# B&R Automation Studio project PT_KB_V01
Automation Studio 4.12.3.127 SP

## Configuration C50_Terminal

CPU 4PPC50.101E-13A, AutomationRuntime B4.93, Build 4.1.2, Vc V4.73.3

### Hardware
```
4PPC50_101E_13A : 4PPC50.101E-13A v1.2.2.0
  Connector IF2:
    ActivateDevice = 1
    Mode = Manual
    InternetAddress = 10.0.0.205
    SubnetMask = 255.255.254.0
  Connector IF3:
    AssignedOperatingSystem = ARemb
  Connector IF4:
    AssignedOperatingSystem = GPOS
  ConfigurationID = PT_KB_V01_C50_Terminal
  TimerDeviceType = SWIOTIMER
  Cyclic1Duration = 10000
  Cyclic1Tolerance = 10000
  Cyclic2Duration = 20000
  Cyclic2Tolerance = 20000
  Cyclic3Duration = 50000
  Cyclic3Tolerance = 50000
  Cyclic4Duration = 100000
  Cyclic4Tolerance = 100000
  Cyclic5Duration = 200000
  Cyclic5Tolerance = 200000
  Cyclic6Duration = 500000
  Cyclic6Tolerance = 500000
  Cyclic7Duration = 1000000
  Cyclic7Tolerance = 1000000
  Cyclic8Duration = 10000
  Cyclic8Tolerance = 30000000
  FileDevice1
  FileDeviceName1 = USER
  FileDevicePath1 = USER_PATH
  LXTMode = Manual
  LXTInternetAddress = 10.0.0.205
  LXTSubnetmask = 255.255.254.0
  LXTActivateDns = 0
  LXTVisuMode = VNC
  LXTVisuURL = 10.0.0.204:5900
  LXTPasswordVNC = 
  LXTUpdateTrigger = 0
```

## Configuration Config1

CPU 4PPC50.101E-13A, AutomationRuntime B4.93, Build 4.1.2, Vc V4.73.3

### Task classes (Cpu.sw)
```
Cyclic#1 (cycle 10000 us, tolerance 10000 us):
  IO <- IO.prg
Cyclic#4 (cycle 100000 us, tolerance 100000 us):
  PID_Pu_01 <- PID_Pu_01.prg
  Rad_PG_KB <- Rad_PG_KB.prg
  PG_Intf <- PG_Intf.prg
  HMI_Svc <- HMI_Svc.prg
  ProcUnit <- ProcessUnit.ProcUnit.prg
  DeviceCtrl <- DeviceCtrl.prg
Cyclic#5 (cycle 200000 us, tolerance 200000 us):
  BRB2_com <- IMA_comm_PG_BRB2.BRB2_com.prg
DataObjects: BRB2 <- IMA_comm_PG_BRB2.BRB2.dob
VcDataObjects: Visu1 <- Visu1.dob
Binaries: vcmgr, arialbd, udbdef, vcpdsw, vcalarm, vcshared, vcgclass, Visu101, vctcal, vccshape, vcnet, TCData, vcpdvnc, vcctext, FWRules, vcdsint, vcfile, Visu102, vcrt, vcbclass, vcpfgen, vcfntttf, vcdsloc, vccovl, Visu103, arial, vccnum, vccstr, vccbtn, ashwd, ashwac, User, sysconf, asfw, arconfig, iomap, Role
Libraries: standard, MTBasics, brsystem, sys_lib, MTTypes, runtime, MTFilter, FileIO, AsArLog, AsArProf, AsMem, DataObj, astime, BR_Lib, VFD_Lib, vcresman, asieccon, AsIMA, inaclnt
```

### Hardware
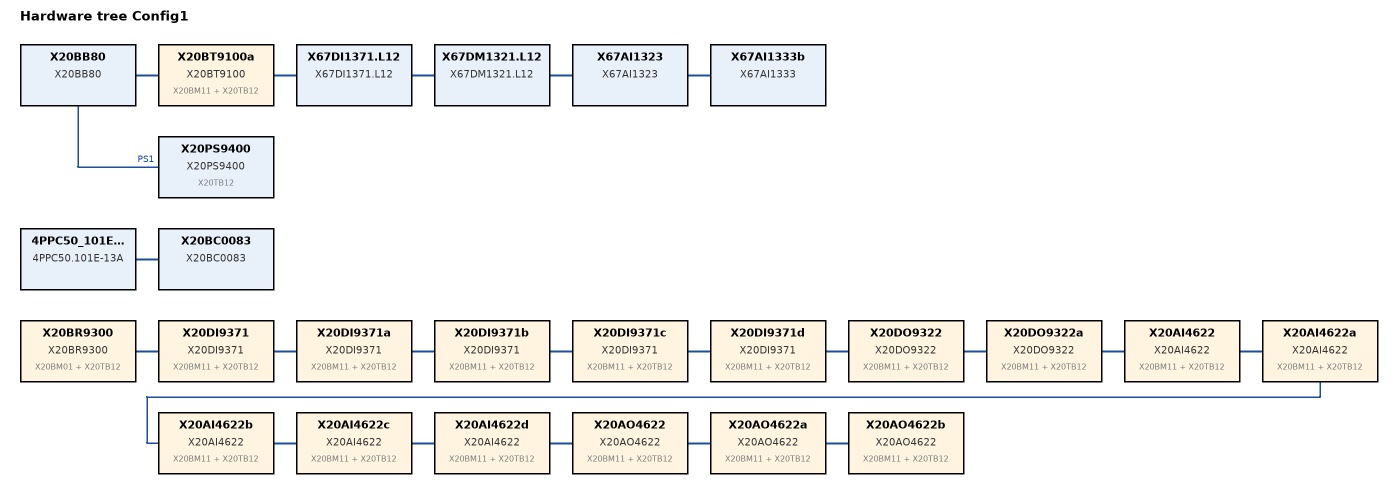
```
4PPC50_101E_13A : 4PPC50.101E-13A v1.2.2.0
  Connector IF2:
    ActivateDevice = 1
    Mode = Manual
    InternetAddress = 10.0.0.204
    SubnetMask = 255.255.254.0
  Connector IF3:
    AssignedOperatingSystem = ARemb
  Connector IF4:
    AssignedOperatingSystem = GPOS
  ConfigurationID = PT_KB_V01_Config1
  RemanentGlobalPvSize = 5000
  VolatileGlobalPvSize = 655350
  RebootReset = 1
  TimerDeviceType = SWIOTIMER
  Cyclic1Duration = 10000
  Cyclic1Tolerance = 10000
  Cyclic2Duration = 20000
  Cyclic2Tolerance = 20000
  Cyclic3Duration = 50000
  Cyclic3Tolerance = 50000
  Cyclic4Duration = 100000
  Cyclic4Tolerance = 100000
  Cyclic5Duration = 200000
  Cyclic5Tolerance = 200000
  Cyclic6Duration = 500000
  Cyclic6Tolerance = 500000
  Cyclic7Duration = 1000000
  Cyclic7Tolerance = 1000000
  Cyclic8Duration = 10000
  Cyclic8Tolerance = 30000000
  FileDevice1
  FileDeviceName1 = USER
  FileDevicePath1 = USER_PATH
  VncVcObjectName = Visu1
  VncMaxConnections = 5
  LXTMode = Manual
  LXTInternetAddress = 10.0.0.205
  LXTSubnetmask = 255.255.254.0
  LXTActivateBuzzer = 1
  LXTVisuMode = VNC
  LXTVisuURL = 10.0.0.204:5900
  LXTPasswordVNC = 
  LXTLocalScaling = 1
  LXTUpdateTrigger = 0
X20AI4622 : X20AI4622 v1.5.0.0  [SS1 -> X20TB12h.SS; SL -> X20BM11g.SL1]
  ChannelType01 = 4 to 20mA
  ChannelType02 = 4 to 20mA
  ChannelType03 = 4 to 20mA
  ChannelType04 = 4 to 20mA
X20AI4622a : X20AI4622 v1.5.0.0  [SS1 -> X20TB12i.SS; SL -> X20BM11h.SL1]
  ChannelType01 = 4 to 20mA
  ChannelType02 = 4 to 20mA
  ChannelType03 = 4 to 20mA
  ChannelType04 = 4 to 20mA
X20AI4622b : X20AI4622 v1.5.0.0  [SS1 -> X20TB12j.SS; SL -> X20BM11i.SL1]
  ChannelType01 = 4 to 20mA
  ChannelType02 = 4 to 20mA
  ChannelType03 = 4 to 20mA
  ChannelType04 = 4 to 20mA
X20AI4622c : X20AI4622 v1.5.0.0  [SS1 -> X20TB12k.SS; SL -> X20BM11j.SL1]
  ChannelType01 = 4 to 20mA
  ChannelType02 = 4 to 20mA
  ChannelType03 = 4 to 20mA
  ChannelType04 = 4 to 20mA
X20AI4622d : X20AI4622 v1.5.0.0  [SS1 -> X20TB12l.SS; SL -> X20BM11k.SL1]
  ChannelType01 = 4 to 20mA
  ChannelType02 = 4 to 20mA
  ChannelType03 = 4 to 20mA
  ChannelType04 = 4 to 20mA
X20AO4622 : X20AO4622 v1.4.1.0  [SS1 -> X20TB12m.SS; SL -> X20BM11l.SL1]
  ChannelType01 = 4 to 20mA
  ChannelType02 = 4 to 20mA
  ChannelType03 = 4 to 20mA
  ChannelType04 = 4 to 20mA
X20AO4622a : X20AO4622 v1.4.1.0  [SS1 -> X20TB12n.SS; SL -> X20BM11m.SL1]
  ChannelType01 = 4 to 20mA
  ChannelType02 = 4 to 20mA
  ChannelType03 = 4 to 20mA
  ChannelType04 = 4 to 20mA
X20AO4622b : X20AO4622 v1.4.1.0  [SS1 -> X20TB12o.SS; SL -> X20BM11n.SL1]
  ChannelType01 = 4 to 20mA
  ChannelType02 = 4 to 20mA
  ChannelType03 = 4 to 20mA
  ChannelType04 = 4 to 20mA
X20BB80 : X20BB80 v1.1.0.0
X20BC0083 : X20BC0083 v2.14.0.0  [PLK1 -> 4PPC50_101E_13A.IF1 (NodeNumber=16) [Cable Type=PowerlinkCable, Length=10, Version=1.0.0.3]; SL -> X20BB80.SL1]
  Supervision = off
X20BM01 : X20BM01 v2.2.0.0
X20BM11 : X20BM11 v1.1.0.0  [X2X1 -> X20BM01.X2X2]
X20BM11a : X20BM11 v1.1.0.0  [X2X1 -> X20BM11.X2X2]
X20BM11b : X20BM11 v1.1.0.0  [X2X1 -> X20BM11a.X2X2]
X20BM11c : X20BM11 v1.1.0.0  [X2X1 -> X20BM11b.X2X2]
X20BM11d : X20BM11 v1.1.0.0  [X2X1 -> X20BM11c.X2X2]
X20BM11e : X20BM11 v1.1.0.0  [X2X1 -> X20BM11d.X2X2]
X20BM11f : X20BM11 v1.1.0.0  [X2X1 -> X20BM11e.X2X2]
X20BM11g : X20BM11 v1.1.0.0  [X2X1 -> X20BM11f.X2X2]
X20BM11h : X20BM11 v1.1.0.0  [X2X1 -> X20BM11g.X2X2]
X20BM11i : X20BM11 v1.1.0.0  [X2X1 -> X20BM11h.X2X2]
X20BM11j : X20BM11 v1.1.0.0  [X2X1 -> X20BM11i.X2X2]
X20BM11k : X20BM11 v1.1.0.0  [X2X1 -> X20BM11j.X2X2]
X20BM11l : X20BM11 v1.1.0.0  [X2X1 -> X20BM11k.X2X2]
X20BM11m : X20BM11 v1.1.0.0  [X2X1 -> X20BM11l.X2X2]
X20BM11n : X20BM11 v1.1.0.0  [X2X1 -> X20BM11m.X2X2]
X20BM11p : X20BM11 v1.1.0.0  [X2X1 -> X20BB80.IF1]
X20BR9300 : X20BR9300 v1.3.0.0  [SS1 -> X20TB12.SS; SL -> X20BM01.SL1; X2X1 -> 4PPC50_101E_13A.IF5 [Cable Type=X2XCable, Length=10, Version=1.0.0.3]]
X20BT9100a : X20BT9100 v1.3.0.0  [SS1 -> X20TB12q.SS; SL -> X20BM11p.SL1]
X20DI9371 : X20DI9371 v1.6.0.0  [SS1 -> X20TB12a.SS; SL -> X20BM11.SL1]
X20DI9371a : X20DI9371 v1.6.0.0  [SS1 -> X20TB12b.SS; SL -> X20BM11a.SL1]
X20DI9371b : X20DI9371 v1.6.0.0  [SS1 -> X20TB12c.SS; SL -> X20BM11b.SL1]
X20DI9371c : X20DI9371 v1.6.0.0  [SS1 -> X20TB12d.SS; SL -> X20BM11c.SL1]
X20DI9371d : X20DI9371 v1.6.0.0  [SS1 -> X20TB12e.SS; SL -> X20BM11d.SL1]
X20DO9322 : X20DO9322 v1.6.0.0  [SS1 -> X20TB12f.SS; SL -> X20BM11e.SL1]
X20DO9322a : X20DO9322 v1.6.0.0  [SS1 -> X20TB12g.SS; SL -> X20BM11f.SL1]
X20PS9400 : X20PS9400 v1.8.0.0  [SS1 -> X20TB12r.SS; PS -> X20BB80.PS1]
X20TB12 : X20TB12 v1.0.0.0
X20TB12a : X20TB12 v1.0.0.0
X20TB12b : X20TB12 v1.0.0.0
X20TB12c : X20TB12 v1.0.0.0
X20TB12d : X20TB12 v1.0.0.0
X20TB12e : X20TB12 v1.0.0.0
X20TB12f : X20TB12 v1.0.0.0
X20TB12g : X20TB12 v1.0.0.0
X20TB12h : X20TB12 v1.0.0.0
X20TB12i : X20TB12 v1.0.0.0
X20TB12j : X20TB12 v1.0.0.0
X20TB12k : X20TB12 v1.0.0.0
X20TB12l : X20TB12 v1.0.0.0
X20TB12m : X20TB12 v1.0.0.0
X20TB12n : X20TB12 v1.0.0.0
X20TB12o : X20TB12 v1.0.0.0
X20TB12q : X20TB12 v1.0.0.0
X20TB12r : X20TB12 v1.0.0.0
X67AI1323 : X67AI1323 v1.1.0.0  [X2X1 -> X67DM1321.L12.X2X2 [Cable Type=X2XCable, Length=10, Version=1.0.0.3]]
  Supervision = off
  InputFilter = level 128
  EnhChannelConfig = on
  ChannelType01 = 4to20mA
  ChannelType02 = 4to20mA
  ChannelType03 = 4to20mA
  ChannelType04 = 4to20mA
X67AI1333b : X67AI1333 v1.1.0.0  [X2X1 -> X67AI1323.X2X2 [Cable Type=X2XCable, Length=10, Version=1.0.0.3]]
  Supervision = off
  InputFilter = level 128
  ChannelType01 = 4to20mA
  ChannelType02 = 4to20mA
  ChannelType03 = 4to20mA
  ChannelType04 = 4to20mA
X67DI1371.L12 : X67DI1371.L12 v1.1.0.0  [X2X1 -> X20BT9100a.X2X1 [Cable Type=X2XCable, Length=10, Version=1.0.0.3]]
  Supervision = off
X67DM1321.L12 : X67DM1321.L12 v1.3.0.0  [X2X1 -> X67DI1371.L12.X2X2 [Cable Type=X2XCable, Length=10, Version=1.0.0.3]]
  Supervision = off
```

### IoMap.iom - 4PPC50_101E_13A/IoMap.iom
```iecst
VAR_CONFIG
	Cyclic#1.PG.Sens.Pt._1.AI_Input.RawValue AT %IW."X20AI4622".AnalogInput01; (* PT01 - pritisak termalne vode na ulazu podstanice [bar]. *)
	Cyclic#1.PG.Sens.Pt._2.AI_Input.RawValue AT %IW."X20AI4622".AnalogInput02; (* PT02 - pritisak posle streinera grubih filtera [bar]. *)
	Cyclic#1.PG.Sens.Pt._3.AI_Input.RawValue AT %IW."X20AI4622".AnalogInput03; (* PT03 - pritisak posle velikog razmenjivaca [bar]. *)
	Cyclic#1.PG.Sens.Pt._4.AI_Input.RawValue AT %IW."X20AI4622".AnalogInput04; (* PT04 - pritisak na ulazu u prihvatni tank [bar]. *)
	Cyclic#1.PG.Sens.Pt._5.AI_Input.RawValue AT %IW."X20AI4622a".AnalogInput01; (* PT05 - pritisak na potisu transportnih pumpi [bar]. *)
	Cyclic#1.PG.Sens.Pt._NS1.AI_Input.RawValue AT %IW."X20AI4622a".AnalogInput02; (* PTNS01 - pritisak na dnu prihvatnog tanka [bar]. *)
	Cyclic#1.PG.Sens.Pt._NS2.AI_Input.RawValue AT %IW."X20AI4622a".AnalogInput03; (* PTNS02 - pritisak na vrhu prihvatnog tanka [bar]. *)
	Cyclic#1.PG.Sens.Pt._0_0.AI_Input.RawValue AT %IW."X20AI4622a".AnalogInput04; (* Pritisak komprimovanog vazduha [bar]. *)
	Cyclic#1.PG.Sens.Tt._7.AI_Input.RawValue AT %IW."X20AI4622b".AnalogInput01;
	Cyclic#1.PG.Sens.Tt._2.AI_Input.RawValue AT %IW."X20AI4622b".AnalogInput02; (* TT_PG_02 - ulaz u prihvatni tank. *)
	Cyclic#1.PG.Sens.Tt._3.AI_Input.RawValue AT %IW."X20AI4622b".AnalogInput03; (* TT_PG_03 - temperatura u prihvatnom tanku. *)
	Cyclic#1.PG.Act.PV._5.PV_Input.AI_Raw AT %IW."X20AI4622b".AnalogInput04; (* PG_PV05 - analogna povratna pozicija ventila. *)
	Cyclic#1.PG.Sens.MP._1.AI_Input.RawValue AT %IW."X20AI4622c".AnalogInput01; (* MP01 - protok potisa ka potrosacima [l/s]. *)
	Cyclic#1.PG.Sens.Pt._6.AI_Input.RawValue AT %IW."X20AI4622c".AnalogInput02; (* PT06 - dodatni transmiter pritiska [bar]. *)
	Cyclic#1.PG.Act.PV._1.PV_Input.AI_Raw AT %IW."X20AI4622d".AnalogInput01; (* PG_PV01 - analogna povratna pozicija ulaznog ventila tanka. *)
	Cyclic#1.PG.Act.PV._2.PV_Input.AI_Raw AT %IW."X20AI4622d".AnalogInput02; (* PG_PV02 - analogna povratna pozicija ulaznog ventila tanka. *)
	Cyclic#1.PG.Act.PV._3.PV_Input.AI_Raw AT %IW."X20AI4622d".AnalogInput03; (* PV03 - analogna povratna pozicija odzracnog ventila ulaza podstanice. *)
	Cyclic#1.PG.Act.PV._4.PV_Input.AI_Raw AT %IW."X20AI4622d".AnalogInput04; (* PV04 - analogna povratna pozicija odzracnog ventila ulaza tanka. *)
	Cyclic#1.PG.Act.Pu._1.mapping.DIO.w_freq AT %QW."X20AO4622".AnalogOutput01; (* PG_Pu01 - frekventni zahtev VFD-a [procenat opsega]. *)
	Cyclic#1.PG.Act.Pu._2.mapping.DIO.w_freq AT %QW."X20AO4622".AnalogOutput02; (* PG_Pu02 - frekventni zahtev VFD-a [procenat opsega]. *)
	Cyclic#1.PG.Act.PV._1.PV_Output.AO_Raw AT %QW."X20AO4622a".AnalogOutput01; (* PG_PV01 - analogna komanda polozaja ulaznog ventila tanka. *)
	Cyclic#1.PG.Act.PV._2.PV_Output.AO_Raw AT %QW."X20AO4622a".AnalogOutput02; (* PG_PV02 - analogna komanda polozaja ulaznog ventila tanka. *)
	Cyclic#1.PG.Act.PV._3.PV_Output.AO_Raw AT %QW."X20AO4622a".AnalogOutput03; (* PV03 - analogna komanda polozaja odzracnog ventila ulaza podstanice. *)
	Cyclic#1.PG.Act.PV._4.PV_Output.AO_Raw AT %QW."X20AO4622a".AnalogOutput04; (* PV04 - analogna komanda polozaja odzracnog ventila ulaza tanka. *)
	Cyclic#1.PG.Act.PV._5.PV_Output.AO_Raw AT %QW."X20AO4622b".AnalogOutput01; (* PG_PV05 - analogna komanda polozaja ventila drenaze/preispiranja. *)
	Cyclic#1.PG.Act.Pu._1.mapping.DIO.r_error AT %IX."X20DI9371".DigitalInput01; (* PG_Pu01 - fault ulaz frekventnog regulatora. *)
	Cyclic#1.PG.Act.Pu._2.mapping.DIO.r_error AT %IX."X20DI9371".DigitalInput02; (* PG_Pu02 - fault ulaz frekventnog regulatora. *)
	Cyclic#1.PG.Act.AV._1.V_Input.CloseFb AT %IX."X20DI9371".DigitalInput03; (* PG_V01 - potvrdjen zatvoren polozaj IEBKB1 dovoda. *)
	Cyclic#1.PG.Act.AV._1.V_Input.OpenFb AT %IX."X20DI9371".DigitalInput04; (* PG_V01 - potvrdjen otvoren polozaj IEBKB1 dovoda. *)
	Cyclic#1.PG.Act.AV._2.V_Input.CloseFb AT %IX."X20DI9371".DigitalInput05; (* PG_V02 - potvrdjen zatvoren polozaj BRB2 dovoda. *)
	Cyclic#1.PG.Act.AV._2.V_Input.OpenFb AT %IX."X20DI9371".DigitalInput06; (* PG_V02 - potvrdjen otvoren polozaj BRB2 dovoda. *)
	Cyclic#1.PG.Act.RV._25.HV_Input.CloseFb AT %IX."X20DI9371b".DigitalInput05; (* PG_RV25 - rucni gasni bypass iz tanka, zatvoren. *)
	Cyclic#1.PG.Act.RV._25.HV_Input.OpenFb AT %IX."X20DI9371b".DigitalInput06; (* PG_RV25 - rucni gasni bypass iz tanka, otvoren. *)
	Cyclic#1.PG.Act.RV._26.HV_Input.CloseFb AT %IX."X20DI9371b".DigitalInput07; (* PG_RV26 - rucni ulazni ventil vakuum pumpe, zatvoren. *)
	Cyclic#1.PG.Act.RV._26.HV_Input.OpenFb AT %IX."X20DI9371b".DigitalInput08; (* PG_RV26 - rucni ulazni ventil vakuum pumpe, otvoren. *)
	Cyclic#1.PG.Act.RV._27.HV_Input.CloseFb AT %IX."X20DI9371b".DigitalInput09; (* PG_RV27 - rucni izlazni ventil vakuum pumpe, zatvoren. *)
	Cyclic#1.PG.Act.RV._27.HV_Input.OpenFb AT %IX."X20DI9371b".DigitalInput10; (* PG_RV27 - rucni izlazni ventil vakuum pumpe, otvoren. *)
	Cyclic#1.PG.Sens.LS._1.DI_Input.SensorIn AT %IX."X20DI9371c".DigitalInput01; (* LS01 - nizak nivo prihvatnog tanka. *)
	Cyclic#1.PG.Sens.LS._2.DI_Input.SensorIn AT %IX."X20DI9371c".DigitalInput02; (* LS02 - donji nivo odzracnog cilindra na ulazu podstanice. *)
	Cyclic#1.PG.Sens.LS._3.DI_Input.SensorIn AT %IX."X20DI9371c".DigitalInput03; (* LS03 - gornji nivo odzracnog cilindra na ulazu podstanice. *)
	Cyclic#1.PG.Sens.LS._4.DI_Input.SensorIn AT %IX."X20DI9371c".DigitalInput04; (* LS04 - donji nivo odzracnog cilindra na ulazu tanka. *)
	Cyclic#1.PG.Sens.LS._5.DI_Input.SensorIn AT %IX."X20DI9371c".DigitalInput05; (* LS05 - gornji nivo odzracnog cilindra na ulazu tanka. *)
	Cyclic#1.PG.Sens.MP._1.AI_Input.TransmitterStatus AT %IX."X20DI9371c".DigitalInput06; (* MP01 - status meraca protoka potisa ka potrosacima. *)
	Cyclic#1.PG.Act.AV._1.V_Input.LampOpen AT %IX."X20DI9371c".DigitalInput07; (* PG_V01 - signal pogona dostigao otvoren kraj. *)
	Cyclic#1.PG.Act.AV._1.V_Input.LampClose AT %IX."X20DI9371c".DigitalInput08; (* PG_V01 - signal pogona dostigao zatvoren kraj. *)
	Cyclic#1.PG.Act.AV._2.V_Input.LampOpen AT %IX."X20DI9371c".DigitalInput09; (* PG_V02 - signal pogona dostigao otvoren kraj. *)
	Cyclic#1.PG.Act.AV._2.V_Input.LampClose AT %IX."X20DI9371c".DigitalInput10; (* PG_V02 - signal pogona dostigao zatvoren kraj. *)
	Cyclic#1.PG.Act.AV._1.V_Input.OverTorque AT %IX."X20DI9371c".DigitalInput11; (* PG_V01 - zastita pogona od prevelikog momenta. *)
	Cyclic#1.PG.Act.Pu._1.mapping.DIO.w_run_fwd AT %QX."X20DO9322".DigitalOutput01; (* PG_Pu01 - komanda rad napred. *)
	Cyclic#1.PG.Act.Pu._1.mapping.DIO.w_reset AT %QX."X20DO9322".DigitalOutput02; (* PG_Pu01 - komanda reset greske pogona. *)
	Cyclic#1.PG.Act.Pu._2.mapping.DIO.w_run_fwd AT %QX."X20DO9322".DigitalOutput03; (* PG_Pu02 - komanda rad napred. *)
	Cyclic#1.PG.Act.Pu._2.mapping.DIO.w_reset AT %QX."X20DO9322".DigitalOutput04; (* PG_Pu02 - komanda reset greske pogona. *)
	Cyclic#1.PG.Act.AV._1.V_Output.CmdOpen AT %QX."X20DO9322".DigitalOutput05; (* PG_V01 - komanda otvaranja bistabilnog IEBKB1 dovoda. *)
	Cyclic#1.PG.Act.AV._1.V_Output.CmdClose AT %QX."X20DO9322".DigitalOutput06; (* PG_V01 - komanda zatvaranja bistabilnog IEBKB1 dovoda. *)
	Cyclic#1.PG.Act.AV._2.V_Output.CmdOpen AT %QX."X20DO9322".DigitalOutput07; (* PG_V02 - komanda otvaranja bistabilnog BRB2 dovoda. *)
	Cyclic#1.PG.Act.AV._2.V_Output.CmdClose AT %QX."X20DO9322".DigitalOutput08; (* PG_V02 - komanda zatvaranja bistabilnog BRB2 dovoda. *)
	Cyclic#1.PG.Act.AV._3.V_Output.Cmd AT %QX."X20DO9322".DigitalOutput09; (* PG_V03 - komanda otvaranja pneumatskog ventila izlaza PG_Pu01. *)
	Cyclic#1.PG.Act.AV._4.V_Output.Cmd AT %QX."X20DO9322".DigitalOutput10; (* PG_V04 - komanda otvaranja pneumatskog ventila izlaza PG_Pu02. *)
	Cyclic#1.PG.Act.AV._5.V_Output.Cmd AT %QX."X20DO9322".DigitalOutput11; (* PG_V05 - komanda otvaranja pneumatskog bypass ventila. *)
	Cyclic#1.PG.Act.AV._6.V_Output.Cmd AT %QX."X20DO9322".DigitalOutput12; (* PG_V06 - komanda otvaranja pneumatske grane PG_PV01. *)
	Cyclic#1.PG.Act.AV._7.V_Output.Cmd AT %QX."X20DO9322a".DigitalOutput01; (* PG_V07 - komanda otvaranja pneumatske grane PG_PV02. *)
	Cyclic#1.PG.Sens.Tt._5.AI_Input.RawValue AT %IW."X67AI1323".AnalogInput01;
	Cyclic#1.PG.Sens.Tt._6.AI_Input.RawValue AT %IW."X67AI1323".AnalogInput02;
	Cyclic#1.PG.Sens.Tt._10.AI_Input.RawValue AT %IW."X67AI1323".AnalogInput03;
	Cyclic#1.PG.Sens.Tt._11.AI_Input.RawValue AT %IW."X67AI1323".AnalogInput04;
	Cyclic#1.PG.Sens.Tt._1.AI_Input.RawValue AT %IW."X67AI1333b".AnalogInput01;
	Cyclic#1.PG.Sens.Tt._4.AI_Input.RawValue AT %IW."X67AI1333b".AnalogInput02;
	Cyclic#1.PG.Sens.Tt._9.AI_Input.RawValue AT %IW."X67AI1333b".AnalogInput03;
	Cyclic#1.PG.Sens.Tt._8.AI_Input.RawValue AT %IW."X67AI1333b".AnalogInput04;
	Cyclic#1.PG.Act.AV._3.V_Input.CloseFb AT %IX."X67DI1371.L12".DigitalInput01;
	Cyclic#1.PG.Act.AV._3.V_Input.OpenFb AT %IX."X67DI1371.L12".DigitalInput02;
	Cyclic#1.PG.Act.AV._4.V_Input.CloseFb AT %IX."X67DI1371.L12".DigitalInput03;
	Cyclic#1.PG.Act.AV._4.V_Input.OpenFb AT %IX."X67DI1371.L12".DigitalInput04;
	Cyclic#1.PG.Act.RV._22.HV_Input.CloseFb AT %IX."X67DI1371.L12".DigitalInput05;
	Cyclic#1.PG.Act.RV._22.HV_Input.OpenFb AT %IX."X67DI1371.L12".DigitalInput06;
	Cyclic#1.PG.Act.RV._23.HV_Input.CloseFb AT %IX."X67DI1371.L12".DigitalInput07;
	Cyclic#1.PG.Act.RV._23.HV_Input.OpenFb AT %IX."X67DI1371.L12".DigitalInput08;
	Cyclic#1.PG.Act.RV._24.HV_Input.CloseFb AT %IX."X67DI1371.L12".DigitalInput09;
	Cyclic#1.PG.Act.RV._24.HV_Input.OpenFb AT %IX."X67DI1371.L12".DigitalInput10;
	Cyclic#1.PG.Act.AV._5.V_Input.CloseFb AT %IX."X67DM1321.L12".DigitalInput01;
	Cyclic#1.PG.Act.AV._5.V_Input.OpenFb AT %IX."X67DM1321.L12".DigitalInput02;
	Cyclic#1.PG.Act.AV._6.V_Input.CloseFb AT %IX."X67DM1321.L12".DigitalInput03;
	Cyclic#1.PG.Act.AV._6.V_Input.OpenFb AT %IX."X67DM1321.L12".DigitalInput04;
	Cyclic#1.PG.Act.AV._7.V_Input.CloseFb AT %IX."X67DM1321.L12".DigitalInput05;
	Cyclic#1.PG.Act.AV._7.V_Input.OpenFb AT %IX."X67DM1321.L12".DigitalInput06;
	Cyclic#1.PG.Act.RV._19.HV_Input.CloseFb AT %IX."X67DM1321.L12".DigitalInput07;
	Cyclic#1.PG.Act.RV._19.HV_Input.OpenFb AT %IX."X67DM1321.L12".DigitalInput08;
	Cyclic#1.PG.Act.RV._21.HV_Input.CloseFb AT %IX."X67DM1321.L12".DigitalInput09;
	Cyclic#1.PG.Act.RV._21.HV_Input.OpenFb AT %IX."X67DM1321.L12".DigitalInput10;
	Cyclic#1.PG.Sens.OWF._1.DI_Input.SensorIn AT %IX."X67DM1321.L12".DigitalInput11;
	Cyclic#1.PG.Sens.OWF._2.DI_Input.SensorIn AT %IX."X67DM1321.L12".DigitalInput12;
END_VAR
```

## Configuration Config2

CPU X20CP1382, AutomationRuntime I4.83, Build 4.1.2, Vc V4.73.0

### Task classes (Cpu.sw)
```
Cyclic#1:
  IO <- Project.IO.prg
Cyclic#4:
  Rad_PG_KB <- Project.Rad_PG_KB.prg
  PID_Pu_PT <- Project.PID_Pu_PT.prg
  PG_Intf <- Project.PG_Intf.prg
  HMI_Svc <- Project.HMI_Svc.prg
  ProcUnit <- ProcessUnit.ProcUnit.prg
  DeviceCtrl <- Project.DeviceCtrl.prg
  Cfg2ATV <- CAN.prg
Cyclic#5:
  BRB2_com <- IMA_comm_PG_BRB2.BRB2_com.prg
DataObjects: BRB2 <- IMA_comm_PG_BRB2.BRB2.dob
VcDataObjects: PG1_1 <- Project.PG1_1.dob
Binaries: vcmgr, arialbd, udbdef, vcpdsw, vcalarm, vcshared, vcgclass, Visu101, vctcal, vccshape, vcnet, TCData, vcpdvnc, vcctext, FWRules, vcdsint, vcfile, Visu102, vcrt, vcbclass, vcfntttf, vcdsloc, vccovl, Visu103, arial, vccnum, vccstr, vccbtn, vcpkat, vccdt, vccline, vcctrend, vccbar, vcpfx20, ashwd, ashwac, User, sysconf, asfw, arconfig, iomap, Role, vcpfgen
Libraries: standard, MTBasics, brsystem, sys_lib, MTTypes, runtime, MTFilter, FileIO, AsArLog, AsArProf, AsMem, DataObj, astime, BR_Lib, VFD_Lib, NashCan1, AsIMA, inaclnt, vcresman, asieccon, ashw
```

### Hardware
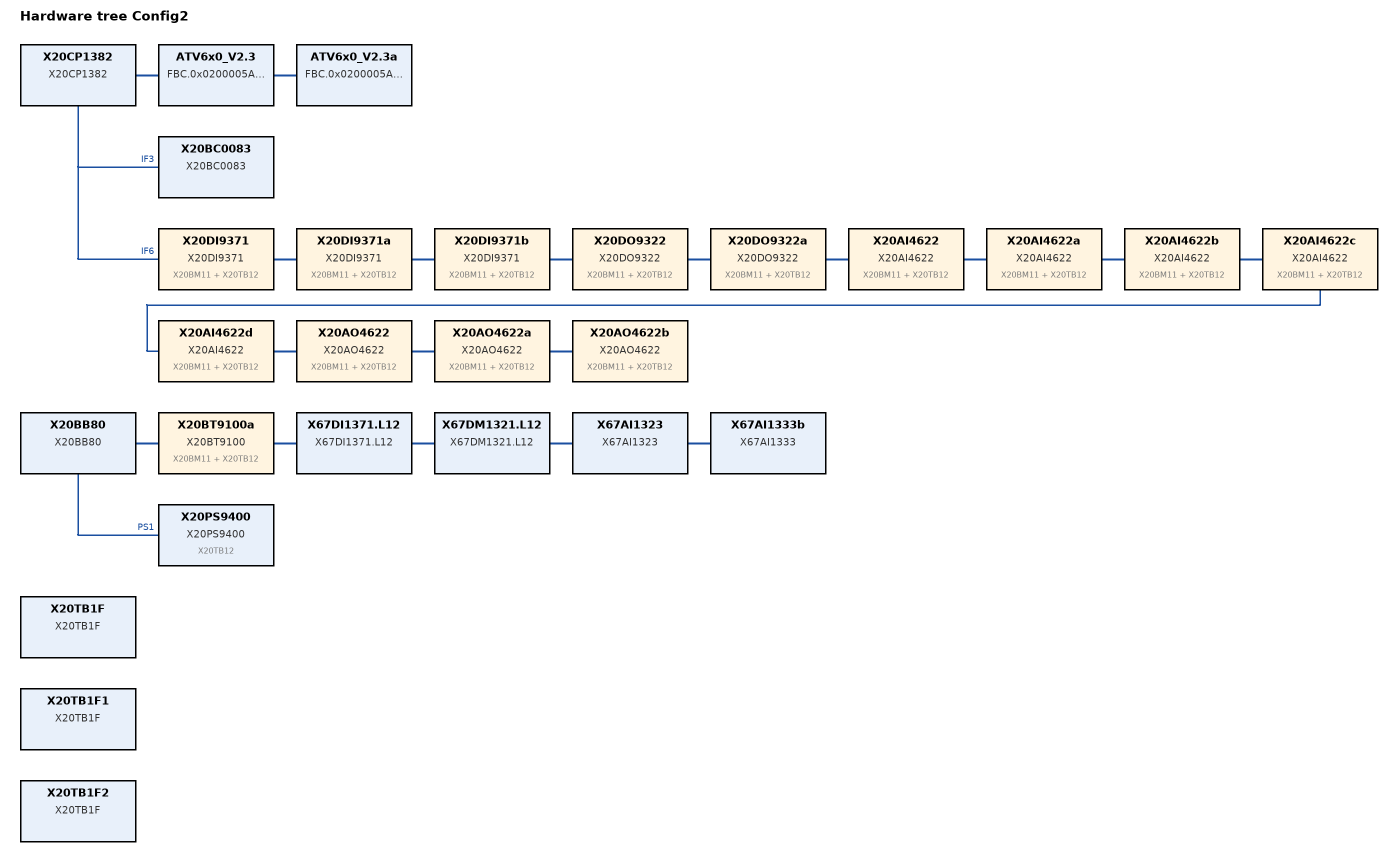
```
ATV6x0_V2.3 : FBC.0x0200005A.600.SEATV6x0_010203E v1.1 (OrderNumber=ATV6x0_V2.3)  [CAN1 -> X20CP1382.IF7 (NodeNumber=3)]
  p2002sub5_connecttomaster = 1
  p2002sub8_connecttomaster = 2
  p2002subc_connecttomaster = 1
  p2061sub2a_connecttomaster = 0
  p2061sub2b_connecttomaster = 0
  p2061sub2c_connecttomaster = 0
  p2061sub2d_connecttomaster = 0
  p2061sub3e_connecttomaster = 0
  p2061sub3f_connecttomaster = 0
  p2061sub40_connecttomaster = 0
  p2061sub41_connecttomaster = 0
  p206bsub30_connecttomaster = 2
  p206bsub31_connecttomaster = 2
  p206bsub32_connecttomaster = 2
  p1801_canidentifier = $NodeID+0x00000280
  pheartbeat_producertime = 100
  p203c_objflags = 1
ATV6x0_V2.3a : FBC.0x0200005A.600.SEATV6x0_010203E v1.1 (OrderNumber=ATV6x0_V2.3)  [CAN1 -> ATV6x0_V2.3.CAN2 (NodeNumber=4)]
  p2002sub5_connecttomaster = 1
  p2002sub8_connecttomaster = 2
  p2002subc_connecttomaster = 1
  p2061sub2a_connecttomaster = 0
  p2061sub2b_connecttomaster = 0
  p2061sub2c_connecttomaster = 0
  p2061sub2d_connecttomaster = 0
  p2061sub3e_connecttomaster = 0
  p2061sub3f_connecttomaster = 0
  p2061sub40_connecttomaster = 0
  p2061sub41_connecttomaster = 0
  p206bsub30_connecttomaster = 2
  p206bsub31_connecttomaster = 2
  p206bsub32_connecttomaster = 2
  p1801_canidentifier = $NodeID+0x00000280
  pheartbeat_producertime = 100
  p203c_objflags = 1
X20AI4622 : X20AI4622 v1.5.0.0  [SS1 -> X20TB12h.SS; SL -> X20BM11g.SL1]
  InputFilter = level 128
  ChannelType01 = 4 to 20mA
  ChannelType02 = 4 to 20mA
  ChannelType03 = 4 to 20mA
  ChannelType04 = 4 to 20mA
X20AI4622a : X20AI4622 v1.5.0.0  [SS1 -> X20TB12i.SS; SL -> X20BM11h.SL1]
  InputFilter = level 128
  ChannelType01 = 4 to 20mA
  ChannelType02 = 4 to 20mA
  ChannelType03 = 4 to 20mA
  ChannelType04 = 4 to 20mA
X20AI4622b : X20AI4622 v1.5.0.0  [SS1 -> X20TB12j.SS; SL -> X20BM11i.SL1]
  InputFilter = level 128
  ChannelType01 = 4 to 20mA
  ChannelType02 = 4 to 20mA
  ChannelType03 = 4 to 20mA
  ChannelType04 = 4 to 20mA
X20AI4622c : X20AI4622 v1.5.0.0  [SS1 -> X20TB12k.SS; SL -> X20BM11j.SL1]
  InputFilter = level 128
  ChannelType01 = 4 to 20mA
  ChannelType02 = 4 to 20mA
  ChannelType03 = 4 to 20mA
  ChannelType04 = 4 to 20mA
X20AI4622d : X20AI4622 v1.5.0.0  [SS1 -> X20TB12l.SS; SL -> X20BM11k.SL1]
  InputFilter = level 128
  ChannelType01 = 4 to 20mA
  ChannelType02 = 4 to 20mA
  ChannelType03 = 4 to 20mA
  ChannelType04 = 4 to 20mA
X20AO4622 : X20AO4622 v1.4.1.0  [SS1 -> X20TB12m.SS; SL -> X20BM11l.SL1]
  ChannelType01 = 4 to 20mA
  ChannelType02 = 4 to 20mA
  ChannelType03 = 4 to 20mA
  ChannelType04 = 4 to 20mA
X20AO4622a : X20AO4622 v1.4.1.0  [SS1 -> X20TB12n.SS; SL -> X20BM11m.SL1]
  ChannelType01 = 4 to 20mA
  ChannelType02 = 4 to 20mA
  ChannelType03 = 4 to 20mA
  ChannelType04 = 4 to 20mA
X20AO4622b : X20AO4622 v1.4.1.0  [SS1 -> X20TB12o.SS; SL -> X20BM11n.SL1]
  ChannelType01 = 4 to 20mA
  ChannelType02 = 4 to 20mA
  ChannelType03 = 4 to 20mA
  ChannelType04 = 4 to 20mA
X20BB80 : X20BB80 v1.1.0.0
X20BC0083 : X20BC0083 v2.14.0.0  [PLK1 -> X20CP1382.IF3 (NodeNumber=16) [Cable Type=PowerlinkCable, Length=10, Version=1.0.0.3]; SL -> X20BB80.SL1]
  Supervision = off
X20BM11 : X20BM11 v1.1.0.0  [X2X1 -> X20CP1382.IF6]
X20BM11b : X20BM11 v1.1.0.0  [X2X1 -> X20BM11.X2X2]
X20BM11c : X20BM11 v1.1.0.0  [X2X1 -> X20BM11b.X2X2]
X20BM11e : X20BM11 v1.1.0.0  [X2X1 -> X20BM11c.X2X2]
X20BM11f : X20BM11 v1.1.0.0  [X2X1 -> X20BM11e.X2X2]
X20BM11g : X20BM11 v1.1.0.0  [X2X1 -> X20BM11f.X2X2]
X20BM11h : X20BM11 v1.1.0.0  [X2X1 -> X20BM11g.X2X2]
X20BM11i : X20BM11 v1.1.0.0  [X2X1 -> X20BM11h.X2X2]
X20BM11j : X20BM11 v1.1.0.0  [X2X1 -> X20BM11i.X2X2]
X20BM11k : X20BM11 v1.1.0.0  [X2X1 -> X20BM11j.X2X2]
X20BM11l : X20BM11 v1.1.0.0  [X2X1 -> X20BM11k.X2X2]
X20BM11m : X20BM11 v1.1.0.0  [X2X1 -> X20BM11l.X2X2]
X20BM11n : X20BM11 v1.1.0.0  [X2X1 -> X20BM11m.X2X2]
X20BM11p : X20BM11 v1.1.0.0  [X2X1 -> X20BB80.IF1]
X20BT9100a : X20BT9100 v1.3.0.0  [SS1 -> X20TB12q.SS; SL -> X20BM11p.SL1]
X20CP1382 : X20CP1382 v1.15.0.0  [X1 -> X1.SL; X2 -> X2.SL; X3 -> X3.SL]
  Module X1 (Type=X1, Virtual=true, Version=1.15.0.0)
    Connection (Connector=SS1, TargetModule=X20TB1F, TargetConnector=SS)
    Connection (Connector=SL, TargetModule=X20CP1382, TargetConnector=X1)
  Module X2 (Type=X2, Virtual=true, Version=1.15.0.0)
    Connection (Connector=SS1, TargetModule=X20TB1F1, TargetConnector=SS)
    Connection (Connector=SL, TargetModule=X20CP1382, TargetConnector=X2)
  Module X3 (Type=X3, Virtual=true, Version=1.15.0.0)
    Connection (Connector=SS1, TargetModule=X20TB1F2, TargetConnector=SS)
    Connection (Connector=SL, TargetModule=X20CP1382, TargetConnector=X3)
  Connector IF2:
    ActivateDevice = 1
    Mode = Manual
    InternetAddress = 10.0.0.204
    SubnetMask = 255.255.254.0
    Vnc1
    VncVcObjectName1 = PG1_1
    VncKeyMappingFile1 = VC\PS2-Keyboard.dis
    VncMaxConnections1 = 10
  Connector IF7:
    ActivateCANIO = 0
    ActivateCanOpen = 1
    pnmtstartup_bit1 = 1
    p100c_parametervalue = 1000
    p100d_parametervalue = 3
  ConfigurationID = PT_KB_V01_Config2
  RemanentGlobalPvSize = 5000
  VolatileGlobalPvSize = 150000
  RebootReset = 1
X20DI9371 : X20DI9371 v1.6.0.0  [SS1 -> X20TB12a.SS; SL -> X20BM11.SL1]
X20DI9371a : X20DI9371 v1.6.0.0  [SS1 -> X20TB12c.SS; SL -> X20BM11b.SL1]
X20DI9371b : X20DI9371 v1.6.0.0  [SS1 -> X20TB12d.SS; SL -> X20BM11c.SL1]
X20DO9322 : X20DO9322 v1.6.0.0  [SS1 -> X20TB12f.SS; SL -> X20BM11e.SL1]
X20DO9322a : X20DO9322 v1.6.0.0  [SS1 -> X20TB12g.SS; SL -> X20BM11f.SL1]
X20PS9400 : X20PS9400 v1.8.0.0  [SS1 -> X20TB12r.SS; PS -> X20BB80.PS1]
X20TB12a : X20TB12 v1.0.0.0
X20TB12c : X20TB12 v1.0.0.0
X20TB12d : X20TB12 v1.0.0.0
X20TB12f : X20TB12 v1.0.0.0
X20TB12g : X20TB12 v1.0.0.0
X20TB12h : X20TB12 v1.0.0.0
X20TB12i : X20TB12 v1.0.0.0
X20TB12j : X20TB12 v1.0.0.0
X20TB12k : X20TB12 v1.0.0.0
X20TB12l : X20TB12 v1.0.0.0
X20TB12m : X20TB12 v1.0.0.0
X20TB12n : X20TB12 v1.0.0.0
X20TB12o : X20TB12 v1.0.0.0
X20TB12q : X20TB12 v1.0.0.0
X20TB12r : X20TB12 v1.0.0.0
X20TB1F : X20TB1F v1.0.0.0
X20TB1F1 : X20TB1F v1.0.0.0
X20TB1F2 : X20TB1F v1.0.0.0
X67AI1323 : X67AI1323 v1.1.0.0  [X2X1 -> X67DM1321.L12.X2X2 [Cable Type=X2XCable, Length=10, Version=1.0.0.3]]
  Supervision = off
  InputFilter = level 128
  EnhChannelConfig = on
  ChannelType01 = 4to20mA
  ChannelType02 = 4to20mA
  ChannelType03 = 4to20mA
  ChannelType04 = 4to20mA
X67AI1333b : X67AI1333 v1.1.0.0  [X2X1 -> X67AI1323.X2X2 [Cable Type=X2XCable, Length=10, Version=1.0.0.3]]
  Supervision = off
  InputFilter = level 128
  ChannelType01 = 4to20mA
  ChannelType02 = 4to20mA
  ChannelType03 = 4to20mA
  ChannelType04 = 4to20mA
X67DI1371.L12 : X67DI1371.L12 v1.1.0.0  [X2X1 -> X20BT9100a.X2X1 [Cable Type=X2XCable, Length=10, Version=1.0.0.3]]
  Supervision = off
X67DM1321.L12 : X67DM1321.L12 v1.3.0.0  [X2X1 -> X67DI1371.L12.X2X2 [Cable Type=X2XCable, Length=10, Version=1.0.0.3]]
  Supervision = off
```

### IoMap.iom - X20CP1382/IoMap.iom
```iecst
VAR_CONFIG
	PT_Alarm.IO.X20AI4622.ModuleOk AT %IX."X20AI4622".ModuleOk;
	PT_Alarm.IO.X20AI4622a.ModuleOk AT %IX."X20AI4622a".ModuleOk;
	PT_Alarm.IO.X20AI4622b.ModuleOk AT %IX."X20AI4622b".ModuleOk;
	PT_Alarm.IO.X20AI4622c.ModuleOk AT %IX."X20AI4622c".ModuleOk;
	PT_Alarm.IO.X20AI4622d.ModuleOk AT %IX."X20AI4622d".ModuleOk;
	PT_Alarm.IO.X20AO4622.ModuleOk AT %IX."X20AO4622".ModuleOk;
	PT_Alarm.IO.X20AO4622a.ModuleOk AT %IX."X20AO4622a".ModuleOk;
	PT_Alarm.IO.X20AO4622b.ModuleOk AT %IX."X20AO4622b".ModuleOk;
	PT_Alarm.IO.X20DI9371.ModuleOk AT %IX."X20DI9371".ModuleOk;
	PT_Alarm.IO.X20DI9371a.ModuleOk AT %IX."X20DI9371a".ModuleOk;
	PT_Alarm.IO.X20DI9371b.ModuleOk AT %IX."X20DI9371b".ModuleOk;
	PT_Alarm.IO.X20DO9322.ModuleOk AT %IX."X20DO9322".ModuleOk;
	PT_Alarm.IO.X20DO9322a.ModuleOk AT %IX."X20DO9322a".ModuleOk;
	PT_Alarm.IO.X20BC0083.ModuleOk AT %IX."X20BC0083".ModuleOk;
	PT_Alarm.IO.X20PS9400.ModuleOk AT %IX."X20PS9400".ModuleOk;
	PT_Alarm.IO.X20BT9100a.ModuleOk AT %IX."X20BT9100a".ModuleOk;
	PT_Alarm.IO.X67AI1323.ModuleOk AT %IX."X67AI1323".ModuleOk;
	PT_Alarm.IO.X67AI1333b.ModuleOk AT %IX."X67AI1333b".ModuleOk;
	PT_Alarm.IO.X67DI1371_L12.ModuleOk AT %IX."X67DI1371.L12".ModuleOk;
	PT_Alarm.IO.X67DM1321_L12.ModuleOk AT %IX."X67DM1321.L12".ModuleOk;
	Cyclic#4.PG.Act.Pu._1.CAN_FB.AtvCanOut.w_ZadataBrz AT %QW."ATV6x0_V2.3".TargetVelocity_6042_Out; (* PG_Pu01 - CANopen zadata brzina ATV630. *)
	Cyclic#4.PG.Act.Pu._1.CAN_FB.AtvCanOut.w_ControlReg AT %QW."ATV6x0_V2.3".Controlword_6040_Out; (* PG_Pu01 - CANopen kontrolna rec ATV630. *)
	Cyclic#4.PG.Act.Pu._1.CAN_FB.AtvCanIn.w_StatusReg AT %IW."ATV6x0_V2.3".Statusword_6041; (* PG_Pu01 - CANopen statusna rec ATV630. *)
	Cyclic#4.PG.Act.Pu._1.CAN_FB.AtvCanIn.w_MotorBrz AT %IW."ATV6x0_V2.3".ControlEffort_6044; (* PG_Pu01 - ostvarena brzina ATV630. *)
	Cyclic#4.PG.Act.Pu._1.CAN_FB.AtvCanIn.w_MotorSnaga AT %IW."ATV6x0_V2.3".OPR_3211_2002subc; (* PG_Pu01 - ostvarena snaga ATV630. *)
	Cyclic#4.PG.Act.Pu._1.CAN_FB.AtvCanIn.w_MotorStruja AT %IW."ATV6x0_V2.3".LCR_3204_2002sub5; (* PG_Pu01 - struja motora ATV630. *)
	Cyclic#4.PG.Act.Pu._1.CAN_FB.AtvCanIn.b_NodeState AT %IX."ATV6x0_V2.3".ModuleOk; (* PG_Pu01 - status CANopen uredjaja. *)
	Cyclic#4.PG.Act.Pu._2.CAN_FB.AtvCanOut.w_ZadataBrz AT %QW."ATV6x0_V2.3a".TargetVelocity_6042_Out; (* PG_Pu02 - CANopen zadata brzina ATV630. *)
	Cyclic#4.PG.Act.Pu._2.CAN_FB.AtvCanOut.w_ControlReg AT %QW."ATV6x0_V2.3a".Controlword_6040_Out; (* PG_Pu02 - CANopen kontrolna rec ATV630. *)
	Cyclic#4.PG.Act.Pu._2.CAN_FB.AtvCanIn.w_StatusReg AT %IW."ATV6x0_V2.3a".Statusword_6041; (* PG_Pu02 - CANopen statusna rec ATV630. *)
	Cyclic#4.PG.Act.Pu._2.CAN_FB.AtvCanIn.w_MotorBrz AT %IW."ATV6x0_V2.3a".ControlEffort_6044; (* PG_Pu02 - ostvarena brzina ATV630. *)
	Cyclic#4.PG.Act.Pu._2.CAN_FB.AtvCanIn.w_MotorSnaga AT %IW."ATV6x0_V2.3a".OPR_3211_2002subc; (* PG_Pu02 - ostvarena snaga ATV630. *)
	Cyclic#4.PG.Act.Pu._2.CAN_FB.AtvCanIn.w_MotorStruja AT %IW."ATV6x0_V2.3a".LCR_3204_2002sub5; (* PG_Pu02 - struja motora ATV630. *)
	Cyclic#4.PG.Act.Pu._2.CAN_FB.AtvCanIn.b_NodeState AT %IX."ATV6x0_V2.3a".ModuleOk; (* PG_Pu02 - status CANopen uredjaja. *)
	Cyclic#1.PG.Sens.Pt._1.AI_Input.RawValue AT %IW."X20AI4622".AnalogInput01; (* PT01 - pritisak termalne vode na ulazu podstanice [bar]. *)
	Cyclic#1.PG.Sens.Pt._2.AI_Input.RawValue AT %IW."X20AI4622".AnalogInput02; (* PT02 - pritisak posle streinera grubih filtera [bar]. *)
	Cyclic#1.PG.Sens.Pt._3.AI_Input.RawValue AT %IW."X20AI4622".AnalogInput03; (* PT03 - pritisak posle velikog razmenjivaca [bar]. *)
	Cyclic#1.PG.Sens.Pt._4.AI_Input.RawValue AT %IW."X20AI4622".AnalogInput04; (* PT04 - pritisak na ulazu u prihvatni tank [bar]. *)
	Cyclic#1.PG.Sens.Pt._5.AI_Input.RawValue AT %IW."X20AI4622a".AnalogInput01; (* PT05 - pritisak na potisu transportnih pumpi [bar]. *)
	Cyclic#1.PG.Sens.Pt._NS1.AI_Input.RawValue AT %IW."X20AI4622a".AnalogInput02; (* PTNS01 - pritisak na dnu prihvatnog tanka [bar]. *)
	Cyclic#1.PG.Sens.Pt._NS2.AI_Input.RawValue AT %IW."X20AI4622a".AnalogInput03; (* PTNS02 - pritisak na vrhu prihvatnog tanka [bar]. *)
	Cyclic#1.PG.Sens.Pt._0_0.AI_Input.RawValue AT %IW."X20AI4622a".AnalogInput04; (* Pritisak komprimovanog vazduha [bar]. *)
	Cyclic#1.PG.Sens.Tt._7.AI_Input.RawValue AT %IW."X20AI4622b".AnalogInput01;
	Cyclic#1.PG.Sens.Tt._2.AI_Input.RawValue AT %IW."X20AI4622b".AnalogInput02; (* TT_PG_02 - ulaz u prihvatni tank. *)
	Cyclic#1.PG.Sens.Tt._3.AI_Input.RawValue AT %IW."X20AI4622b".AnalogInput03; (* TT_PG_03 - temperatura u prihvatnom tanku. *)
	Cyclic#1.PG.Act.PV._5.PV_Input.AI_Raw AT %IW."X20AI4622b".AnalogInput04; (* PG_PV05 - analogna povratna pozicija ventila. *)
	Cyclic#1.PG.Sens.MP._1.AI_Input.RawValue AT %IW."X20AI4622c".AnalogInput01; (* MP01 - protok potisa ka potrosacima [l/s]. *)
	Cyclic#1.PG.Sens.Pt._6.AI_Input.RawValue AT %IW."X20AI4622c".AnalogInput02; (* PT06 - dodatni transmiter pritiska [bar]. *)
	Cyclic#1.PG.Act.PV._1.PV_Input.AI_Raw AT %IW."X20AI4622d".AnalogInput01; (* PG_PV01 - analogna povratna pozicija ulaznog ventila tanka. *)
	Cyclic#1.PG.Act.PV._2.PV_Input.AI_Raw AT %IW."X20AI4622d".AnalogInput02; (* PG_PV02 - analogna povratna pozicija ulaznog ventila tanka. *)
	Cyclic#1.PG.Act.PV._3.PV_Input.AI_Raw AT %IW."X20AI4622d".AnalogInput03; (* PV03 - analogna povratna pozicija odzracnog ventila ulaza podstanice. *)
	Cyclic#1.PG.Act.PV._4.PV_Input.AI_Raw AT %IW."X20AI4622d".AnalogInput04; (* PV04 - analogna povratna pozicija odzracnog ventila ulaza tanka. *)
	Cyclic#1.PG.Act.PV._1.PV_Output.AO_Raw AT %QW."X20AO4622a".AnalogOutput01; (* PG_PV01 - analogna komanda polozaja ulaznog ventila tanka. *)
	Cyclic#1.PG.Act.PV._2.PV_Output.AO_Raw AT %QW."X20AO4622a".AnalogOutput02; (* PG_PV02 - analogna komanda polozaja ulaznog ventila tanka. *)
	Cyclic#1.PG.Act.PV._3.PV_Output.AO_Raw AT %QW."X20AO4622a".AnalogOutput03; (* PV03 - analogna komanda polozaja odzracnog ventila ulaza podstanice. *)
	Cyclic#1.PG.Act.PV._4.PV_Output.AO_Raw AT %QW."X20AO4622a".AnalogOutput04; (* PV04 - analogna komanda polozaja odzracnog ventila ulaza tanka. *)
	Cyclic#1.PG.Act.PV._5.PV_Output.AO_Raw AT %QW."X20AO4622b".AnalogOutput01; (* PG_PV05 - analogna komanda polozaja ventila drenaze/preispiranja. *)
	Cyclic#1.PG.Act.AV._1.V_Input.CloseFb AT %IX."X20DI9371".DigitalInput03; (* PG_V01 - potvrdjen zatvoren polozaj IEBKB1 dovoda. *)
	Cyclic#1.PG.Act.AV._1.V_Input.OpenFb AT %IX."X20DI9371".DigitalInput04; (* PG_V01 - potvrdjen otvoren polozaj IEBKB1 dovoda. *)
	Cyclic#1.PG.Act.AV._2.V_Input.CloseFb AT %IX."X20DI9371".DigitalInput05; (* PG_V02 - potvrdjen zatvoren polozaj BRB2 dovoda. *)
	Cyclic#1.PG.Act.AV._2.V_Input.OpenFb AT %IX."X20DI9371".DigitalInput06; (* PG_V02 - potvrdjen otvoren polozaj BRB2 dovoda. *)
	Cyclic#1.PG.Act.RV._25.HV_Input.CloseFb AT %IX."X20DI9371a".DigitalInput05; (* PG_RV25 - rucni gasni bypass iz tanka, zatvoren. *)
	Cyclic#1.PG.Act.RV._25.HV_Input.OpenFb AT %IX."X20DI9371a".DigitalInput06; (* PG_RV25 - rucni gasni bypass iz tanka, otvoren. *)
	Cyclic#1.PG.Act.RV._26.HV_Input.CloseFb AT %IX."X20DI9371a".DigitalInput07; (* PG_RV26 - rucni ulazni ventil vakuum pumpe, zatvoren. *)
	Cyclic#1.PG.Act.RV._26.HV_Input.OpenFb AT %IX."X20DI9371a".DigitalInput08; (* PG_RV26 - rucni ulazni ventil vakuum pumpe, otvoren. *)
	Cyclic#1.PG.Act.RV._27.HV_Input.CloseFb AT %IX."X20DI9371a".DigitalInput09; (* PG_RV27 - rucni izlazni ventil vakuum pumpe, zatvoren. *)
	Cyclic#1.PG.Act.RV._27.HV_Input.OpenFb AT %IX."X20DI9371a".DigitalInput10; (* PG_RV27 - rucni izlazni ventil vakuum pumpe, otvoren. *)
	Cyclic#1.PG.Sens.LS._1.DI_Input.SensorIn AT %IX."X20DI9371b".DigitalInput01; (* LS01 - nizak nivo prihvatnog tanka. *)
	Cyclic#1.PG.Sens.LS._2.DI_Input.SensorIn AT %IX."X20DI9371b".DigitalInput02; (* LS02 - donji nivo odzracnog cilindra na ulazu podstanice. *)
	Cyclic#1.PG.Sens.LS._3.DI_Input.SensorIn AT %IX."X20DI9371b".DigitalInput03; (* LS03 - gornji nivo odzracnog cilindra na ulazu podstanice. *)
	Cyclic#1.PG.Sens.LS._4.DI_Input.SensorIn AT %IX."X20DI9371b".DigitalInput04; (* LS04 - donji nivo odzracnog cilindra na ulazu tanka. *)
	Cyclic#1.PG.Sens.LS._5.DI_Input.SensorIn AT %IX."X20DI9371b".DigitalInput05; (* LS05 - gornji nivo odzracnog cilindra na ulazu tanka. *)
	Cyclic#1.PG.Sens.MP._1.AI_Input.TransmitterStatus AT %IX."X20DI9371b".DigitalInput06; (* MP01 - status meraca protoka potisa ka potrosacima. *)
	Cyclic#1.PG.Act.AV._1.V_Input.LampOpen AT %IX."X20DI9371b".DigitalInput07; (* PG_V01 - signal pogona dostigao otvoren kraj. *)
	Cyclic#1.PG.Act.AV._1.V_Input.LampClose AT %IX."X20DI9371b".DigitalInput08; (* PG_V01 - signal pogona dostigao zatvoren kraj. *)
	Cyclic#1.PG.Act.AV._2.V_Input.LampOpen AT %IX."X20DI9371b".DigitalInput09; (* PG_V02 - signal pogona dostigao otvoren kraj. *)
	Cyclic#1.PG.Act.AV._2.V_Input.LampClose AT %IX."X20DI9371b".DigitalInput10; (* PG_V02 - signal pogona dostigao zatvoren kraj. *)
	Cyclic#1.PG.Act.AV._1.V_Input.OverTorque AT %IX."X20DI9371b".DigitalInput11; (* PG_V01 - zastita pogona od prevelikog momenta. *)
	Cyclic#1.PG.Act.AV._1.V_Output.CmdOpen AT %QX."X20DO9322".DigitalOutput05; (* PG_V01 - komanda otvaranja bistabilnog IEBKB1 dovoda. *)
	Cyclic#1.PG.Act.AV._1.V_Output.CmdClose AT %QX."X20DO9322".DigitalOutput06; (* PG_V01 - komanda zatvaranja bistabilnog IEBKB1 dovoda. *)
	Cyclic#1.PG.Act.AV._2.V_Output.CmdOpen AT %QX."X20DO9322".DigitalOutput07; (* PG_V02 - komanda otvaranja bistabilnog BRB2 dovoda. *)
	Cyclic#1.PG.Act.AV._2.V_Output.CmdClose AT %QX."X20DO9322".DigitalOutput08; (* PG_V02 - komanda zatvaranja bistabilnog BRB2 dovoda. *)
	Cyclic#1.PG.Act.AV._3.V_Output.Cmd AT %QX."X20DO9322".DigitalOutput09; (* PG_V03 - komanda otvaranja pneumatskog ventila izlaza PG_Pu01. *)
	Cyclic#1.PG.Act.AV._4.V_Output.Cmd AT %QX."X20DO9322".DigitalOutput10; (* PG_V04 - komanda otvaranja pneumatskog ventila izlaza PG_Pu02. *)
	Cyclic#1.PG.Act.AV._5.V_Output.Cmd AT %QX."X20DO9322".DigitalOutput11; (* PG_V05 - komanda otvaranja pneumatskog bypass ventila. *)
	Cyclic#1.PG.Act.AV._6.V_Output.Cmd AT %QX."X20DO9322".DigitalOutput12; (* PG_V06 - komanda otvaranja pneumatske grane PG_PV01. *)
	Cyclic#1.PG.Act.AV._7.V_Output.Cmd AT %QX."X20DO9322a".DigitalOutput01; (* PG_V07 - komanda otvaranja pneumatske grane PG_PV02. *)
	Cyclic#1.PG.Sens.Tt._5.AI_Input.RawValue AT %IW."X67AI1323".AnalogInput01;
	Cyclic#1.PG.Sens.Tt._6.AI_Input.RawValue AT %IW."X67AI1323".AnalogInput02;
	Cyclic#1.PG.Sens.Tt._10.AI_Input.RawValue AT %IW."X67AI1323".AnalogInput03;
	Cyclic#1.PG.Sens.Tt._11.AI_Input.RawValue AT %IW."X67AI1323".AnalogInput04;
	Cyclic#1.PG.Sens.Tt._1.AI_Input.RawValue AT %IW."X67AI1333b".AnalogInput01;
	Cyclic#1.PG.Sens.Tt._4.AI_Input.RawValue AT %IW."X67AI1333b".AnalogInput02;
	Cyclic#1.PG.Sens.Tt._9.AI_Input.RawValue AT %IW."X67AI1333b".AnalogInput03;
	Cyclic#1.PG.Sens.Tt._8.AI_Input.RawValue AT %IW."X67AI1333b".AnalogInput04;
	Cyclic#1.PG.Act.AV._3.V_Input.CloseFb AT %IX."X67DI1371.L12".DigitalInput01;
	Cyclic#1.PG.Act.AV._3.V_Input.OpenFb AT %IX."X67DI1371.L12".DigitalInput02;
	Cyclic#1.PG.Act.AV._4.V_Input.CloseFb AT %IX."X67DI1371.L12".DigitalInput03;
	Cyclic#1.PG.Act.AV._4.V_Input.OpenFb AT %IX."X67DI1371.L12".DigitalInput04;
	Cyclic#1.PG.Act.RV._22.HV_Input.CloseFb AT %IX."X67DI1371.L12".DigitalInput05;
	Cyclic#1.PG.Act.RV._22.HV_Input.OpenFb AT %IX."X67DI1371.L12".DigitalInput06;
	Cyclic#1.PG.Act.RV._23.HV_Input.CloseFb AT %IX."X67DI1371.L12".DigitalInput07;
	Cyclic#1.PG.Act.RV._23.HV_Input.OpenFb AT %IX."X67DI1371.L12".DigitalInput08;
	Cyclic#1.PG.Act.RV._24.HV_Input.CloseFb AT %IX."X67DI1371.L12".DigitalInput09;
	Cyclic#1.PG.Act.RV._24.HV_Input.OpenFb AT %IX."X67DI1371.L12".DigitalInput10;
	Cyclic#1.PG.Act.AV._5.V_Input.CloseFb AT %IX."X67DM1321.L12".DigitalInput01;
	Cyclic#1.PG.Act.AV._5.V_Input.OpenFb AT %IX."X67DM1321.L12".DigitalInput02;
	Cyclic#1.PG.Act.AV._6.V_Input.CloseFb AT %IX."X67DM1321.L12".DigitalInput03;
	Cyclic#1.PG.Act.AV._6.V_Input.OpenFb AT %IX."X67DM1321.L12".DigitalInput04;
	Cyclic#1.PG.Act.AV._7.V_Input.CloseFb AT %IX."X67DM1321.L12".DigitalInput05;
	Cyclic#1.PG.Act.AV._7.V_Input.OpenFb AT %IX."X67DM1321.L12".DigitalInput06;
	Cyclic#1.PG.Act.RV._19.HV_Input.CloseFb AT %IX."X67DM1321.L12".DigitalInput07;
	Cyclic#1.PG.Act.RV._19.HV_Input.OpenFb AT %IX."X67DM1321.L12".DigitalInput08;
	Cyclic#1.PG.Act.RV._21.HV_Input.CloseFb AT %IX."X67DM1321.L12".DigitalInput09;
	Cyclic#1.PG.Act.RV._21.HV_Input.OpenFb AT %IX."X67DM1321.L12".DigitalInput10;
	Cyclic#1.PG.Sens.OWF._1.DI_Input.SensorIn AT %IX."X67DM1321.L12".DigitalInput11;
	Cyclic#1.PG.Sens.OWF._2.DI_Input.SensorIn AT %IX."X67DM1321.L12".DigitalInput12;
	Cyclic#4.PG.Act.Pu._1.Node_status AT %IW."ATV6x0_V2.3".NodeStatus;
	Cyclic#4.PG.Act.Pu._1.U_int.U_srednje AT %IW."ATV6x0_V2.3".ULN_3207_2002sub8;
	Cyclic#4.PG.Act.Pu._1.U_int.U_12 AT %IW."ATV6x0_V2.3".UL1_13747_206bsub30;
	Cyclic#4.PG.Act.Pu._1.U_int.U_23 AT %IW."ATV6x0_V2.3".UL2_13748_206bsub31;
	Cyclic#4.PG.Act.Pu._1.U_int.U_31 AT %IW."ATV6x0_V2.3".UL3_13749_206bsub32;
	Cyclic#4.PG.Act.Pu._2.Node_status AT %IW."ATV6x0_V2.3a".NodeStatus;
	Cyclic#4.PG.Act.Pu._2.U_int.U_srednje AT %IW."ATV6x0_V2.3a".ULN_3207_2002sub8;
	Cyclic#4.PG.Act.Pu._2.U_int.U_12 AT %IW."ATV6x0_V2.3a".UL1_13747_206bsub30;
	Cyclic#4.PG.Act.Pu._2.U_int.U_23 AT %IW."ATV6x0_V2.3a".UL2_13748_206bsub31;
	Cyclic#4.PG.Act.Pu._2.U_int.U_31 AT %IW."ATV6x0_V2.3a".UL3_13749_206bsub32;
END_VAR
```

## Logical view

Binary libraries used (declarations not repeated): operator, runtime, astime, AsIecCon, standard, MTBasics, brsystem, sys_lib, MTTypes, MTFilter 5.16.0, FileIO, AsArLog, AsArProf, AsMem, DataObj, AsIMA, inaclnt

### Global.typ - Global data types
```iecst
TYPE
	PG_type : 	STRUCT  (* Korenski tip objekta: Podstanica grejanja 1, Kursumlijska Banja *)
		Act : PG_Act_type; (* Aktuatori podstanice: pumpe, ventili *)
		Sens : PG_Sens_type; (* Senzori podstanice: pritisak, temperatura, protok, nivo *)
	END_STRUCT;
	PG_Act_type : 	STRUCT  (* Svi aktuatori podstanice PG *)
		Pu : PG_Act_Pu_type; (* Pumpe za snabdevanje potrosaca, Grundfoss CR45, METOD_DIO, 0-50 Hz *)
		PV : PG_Act_PV_type; (* Proporcionalni membranski ventili Burkert, AI/AO 4-20mA *)
		AV : PG_Act_AV_type; (* Automatski leptir ventili End Armaturen DN125 *)
		RV : PG_Act_RV_type; (* Rucni leptir ventili sa 2 krajnja prekidaca, monitoring pozicije *)
	END_STRUCT;
	PG_Sens_type : 	STRUCT  (* Svi senzori podstanice PG *)
		Pt : PG_Sens_Pt_type; (* Senzori pritiska termalne vode, Cerabar PMP23, 4-20mA *)
		Tt : PG_Sens_Tt_type; (* Senzori temperature termalne vode, Easytemp TMR35, 4-20mA *)
		MP : PG_Sens_MP_type; (* Meraci protoka termalne vode, Promag H10, 4-20mA *)
		LS : PG_Sens_LS_type; (* Nivo prekidaci u prihvatnom tanku i odzracnim cilindrima *)
		OWF : PG_Sens_OWF_type; (* Zastitni prestrujni ventili od hidraulickog udara *)
	END_STRUCT;
	PG_Act_Pu_type : 	STRUCT  (* Pumpe za snabdevanje potrosaca + vfdMain FB instance *)
		_1 : VFD_type; (* Pumpa za snabdevanje potrosaca 01, Grundfoss CR45 *)
		_2 : VFD_type; (* Pumpa za snabdevanje potrosaca 02, Grundfoss CR45 *)
		VFD_function : PG_Act_Pu_VFD_func_type; (* vfdMain FB instance za obe pumpe, METOD_DIO *)
	END_STRUCT;
	PG_Act_Pu_VFD_func_type : 	STRUCT  (* vfdMain FB instance za upravljanje frekventnim regulatorima pumpi, 0-50 Hz *)
		_1 : vfdMain; (* vfdMain FB za Pumpu 01, addr_struct inicijalizovan u IO_Init *)
		_2 : vfdMain; (* vfdMain FB za Pumpu 02, addr_struct inicijalizovan u IO_Init *)
	END_STRUCT;
	PG_Act_PV_type : 	STRUCT  (* Proporcionalni membranski ventili Burkert, AI povratni + AO komanda, 4-20mA *)
		_1 : FB_PvAiAo_Fast; (* Ulazni regulacioni ventil 1 - prihvatni tank, DN050 NC *)
		_2 : FB_PvAiAo_Fast; (* Ulazni regulacioni ventil 2 - prihvatni tank, DN050 NC *)
		_3 : FB_PvAiAo_Fast; (* Odzracni ventil na ulazu termalne vode u kotlarnicu, DN025 NC *)
		_4 : FB_PvAiAo_Fast; (* Odzracni ventil na ulazu termalne vode u prihvatni tank, DN025 NC *)
		_5 : FB_PvAiAo_Fast; (* Dodatni proporcionalni ventil, Fast varijanta kao ostali PV kanali *)
	END_STRUCT;
	PG_Act_AV_type : 	STRUCT  (* Automatski leptir ventili End Armaturen DN125, bistabilni i spring-return *)
		_1 : FB_V_EMV; (* Elektromotorni bistabilni, CmdOpen + CmdClose, OpenMaxTime=20s *)
		_2 : FB_V_EMV; (* Elektromotorni bistabilni, CmdOpen + CmdClose, OpenMaxTime=20s *)
		_3 : FB_V_ON_OFF_FB; (* Pneumatski NC spring-return, samo CmdOpen, OpenMaxTime=10s *)
		_4 : FB_V_ON_OFF_FB; (* Pneumatski NC spring-return, samo CmdOpen, OpenMaxTime=10s *)
		_5 : FB_V_ON_OFF_FB; (* Pneumatski NC spring-return, samo CmdOpen, OpenMaxTime=10s *)
		_6 : FB_V_ON_OFF_FB; (* Pneumatski NC spring-return, samo CmdOpen, OpenMaxTime=10s *)
		_7 : FB_V_ON_OFF_FB; (* Pneumatski NC spring-return, samo CmdOpen, OpenMaxTime=10s *)
	END_STRUCT;
	PG_Act_RV_type : 	STRUCT  (* Rucni leptir ventili NIOB FLUID / End Armaturen, monitoring 2 krajnja prekidaca *)
		_19 : FB_HV_2LS; (* Rucni ventil posle membranskog ventila PG_PV01 *)
		_21 : FB_HV_2LS; (* Rucni ventil posle membranskog ventila PG_PV02 *)
		_22 : FB_HV_2LS; (* Drenazni total ventil na dnu prihvatnog tanka *)
		_23 : FB_HV_2LS; (* Ulaz u Pumpu PG_Pu01 *)
		_24 : FB_HV_2LS; (* Ulaz u Pumpu PG_Pu02 *)
		_25 : FB_HV_2LS; (* Bajpasni izlaz iz tanka ka instalaciji za izbacivanje gasa van kotlarnice *)
		_26 : FB_HV_2LS; (* Ulaz u vakuum pumpu *)
		_27 : FB_HV_2LS; (* Izlaz iz vakuum pumpe ka instalaciji za izbacivanje gasa van kotlarnice *)
	END_STRUCT;
	PG_Sens_Pt_type : 	STRUCT  (* Senzori pritiska termalne vode, 9x FBAI01_DI01, Cerabar PMP23, 4-20mA, opseg -1..9 bar / -100..300 mbar / -1..14 bar *)
		_0_0 : FBAI01_DI01; (* Pritisak komprimovanog vazduha, opseg -1..14 bar *)
		_1 : FBAI01_DI01; (* Pritisak termalne vode na ulazu u podstanicu *)
		_2 : FBAI01_DI01; (* Pritisak termalne vode posle streinera grubih filtera *)
		_3 : FBAI01_DI01; (* Pritisak termalne vode posle velikog izmenjivaca *)
		_4 : FBAI01_DI01; (* Pritisak termalne vode na ulazu u prihvatni tank *)
		_5 : FBAI01_DI01; (* Pritisak na potisu transportnih pumpi *)
		_6 : FBAI01_DI01; (* Dodatni transmiter pritiska, opseg -1..9 bar *)
		_NS1 : FBAI01_DI01; (* Pritisak na dnu prihvatnog tanka [mbar] *)
		_NS2 : FBAI01_DI01; (* Pritisak na vrhu prihvatnog tanka [mbar] *)
	END_STRUCT;
	PG_Sens_Tt_type : 	STRUCT  (* Senzori temperature termalne vode, Easytemp TMR35, 4-20mA, opseg 0-120 degC *)
		_1 : FBAI01_DI01; (* TT_PG_01 - ulaz u veliki razmenjivac PGRT01. *)
		_2 : FBAI01_DI01; (* TT_PG_02 - temperatura na ulazu u prihvatni tank. *)
		_3 : FBAI01_DI01; (* TT_PG_03 - temperatura u prihvatnom tanku. *)
		_4 : FBAI01_DI01; (* TT_PG_04 - izlaz iz velikog razmenjivaca PGRT01. *)
		_5 : FBAI01_DI01; (* TT_PG_05 - ulaz u mali razmenjivac PGRT02. *)
		_6 : FBAI01_DI01; (* TT_PG_06 - izlaz iz malog razmenjivaca PGRT02. *)
		_7 : FBAI01_DI01; (* TT_PG_07 - drenazni vod za potvrdu zavrsetka preispiranja. *)
		_8 : FBAI01_DI01; (* TT_PG_08 - Ulaz tehnicke vode u direktni iztmenbjivac toplote*)
		_9 : FBAI01_DI01; (* TT_PG_09 - Izlaz tehnicke vode iz direktnog iztmenbjivaca toplote*)
		_10 : FBAI01_DI01; (* TT_PG_10 - Ulaz tsanitarne vode u direktni iztmenbjivac toplote*)
		_11 : FBAI01_DI01; (* TT_PG_11 - Izlaz sanitarne vode iz direktnog iztmenbjivaca toplote*)
	END_STRUCT;
	PG_Sens_MP_type : 	STRUCT  (* Meraci protoka, 1x FBAI01_DI01, Promag H10 DN065, 4-20mA, opseg 0-72 m3/h *)
		_1 : FBAI01_DI01; (* Merač protoka na potisu tople termalne vode ka potrosacima *)
	END_STRUCT;
	PG_Sens_LS_type : 	STRUCT  (* Nivo prekidaci Liquipoint FTW23, 5x FB_DI, detekcija tecnosti u prihvatnom tanku i odzracnim cilindrima *)
		_1 : FB_DI; (* Nizak nivo vode u prihvatnom tanku za rad pumpi *)
		_2 : FB_DI; (* Donji nivo u odzracnom cilindru na ulazu vode u podstanicu *)
		_3 : FB_DI; (* Gornji nivo u odzracnom cilindru na ulazu vode u podstanicu *)
		_4 : FB_DI; (* Donji nivo u odzracnom cilindru na ulazu vode u prihvatni tank *)
		_5 : FB_DI; (* Gornji nivo u odzracnom cilindru na ulazu vode u prihvatni tank *)
	END_STRUCT;
	PG_Sens_OWF_type : 	STRUCT  (* Zastitni prestrujni ventili NIOB FLUID 5371 DN050, 2x FB_DI, zastita od hidraulickog udara *)
		_1 : FB_DI; (* Zastitni prestrujni ventil od hidraulickog udara 1 *)
		_2 : FB_DI; (* Zastitni prestrujni ventil od hidraulickog udara 2 *)
	END_STRUCT;
	E_PGRad_State :
		( (* Koraci state masine podstanice. *)
		PG_00_Stand_By,
		PG_01_Priprema_BRB2,
		PG_02_Rad_BRB2,
		PG_03_Zaustavljanje_BRB2,
		PG_11_Priprema_IEBKB1,
		PG_12_Rad_IEBKB1,
		PG_13_Zaustavljanje_IEBKB1
		);
	E_RegulacionaVarijanta :
		(
		_00_neaktivan, (* 0 - sve ugaseno, ni jedna varijanta nije izabrana. *)
		_01_REG_PRITISAK, (* 1 - PT vodi, prati zadati pritisak. *)
		_02_REG_NIVO, (* 2 - PT vodi nivo prihvatnog tanka preko izlazne pumpe. *)
		_03_REG_TEMPERATURA (* 3 - temperatura/snaga sekundara. *)
		);
	E_SelektovaniIzvor :
		(
		_00_IZVOR_NIJE_IZABRAN, (* 0 - nijedan izvor nije izabran. *)
		_01_BRB2, (* 1 - BRB2 kao izvor. *)
		_02_IEBKB1 (* 2 - IEBKB1 kao izvor. *)
		);
	E_AktivnaPumpaIzlazTanka :
		(
		_00_nijedna, (* 0 - nijedna pumpa aktivna na izlazu iz tanka. *)
		_01_Pu_PG_01, (* 1 - Pu_PG_01 aktivna. *)
		_02_Pu_PG_02 (* 2 - Pu_PG_02 aktivna. *)
		);
	E_AktivniPropVentilUlazTanka :
		(
		_00_PROP_VENTIL_NIJE_IZABRAN, (* 0 - nijedan prop. ventil nije izabran. *)
		_01_PG_PV01, (* 1 - PG_PV01 aktivan. *)
		_02_PG_PV02 (* 2 - PG_PV02 aktivan. *)
		);
	typCmdRetainUlazniVentiliPGRad : 	STRUCT
		V01_Open : BOOL; (* PG_V01 - zapamceni zahtev IEBKB1 ulaznog ventila. *)
		V02_Open : BOOL; (* PG_V02 - zapamceni zahtev BRB2 ulaznog ventila. *)
	END_STRUCT;
	typParAirReleaseModePGRad : 	STRUCT  (* Parametri odzracivanja za jedan izvor vode. *)
		PV03 : typParAirRelease; (* Odzracivanje na ulazu termalne vode u podstanicu. *)
		PV04 : typParAirRelease; (* Odzracivanje na ulazu termalne vode u prihvatni tank. *)
	END_STRUCT;
	typParAirReleasePGRad : 	STRUCT  (* Grupisani parametri odzracivanja prema aktivnom izvoru. *)
		BRB2 : typParAirReleaseModePGRad; (* Parametri rada sa izvorom BRB2. *)
		IEBKB1 : typParAirReleaseModePGRad; (* Parametri rada sa izvorom IEBKB1. *)
	END_STRUCT;
	typTimeSPPGRad : 	STRUCT  (* Grupisani vremenski SP parametri u sekundama. *)
		PrelazPV05Cuvar_s : REAL; (* Vreme PT06 SP rampe [s]. *)
		OverlapPumpi_s : REAL; (* Maksimalno vreme paralelnog rada pri rotaciji [s]. *)
		AutoRestartDelay_s : REAL; (* Zadrzavanje pre automatskog starta [s]. *)
		ValvePositionTimeout_s : REAL; (* Maksimalno vreme hoda ventila [s]. *)
		InterlockDebounce_s : REAL; (* Vreme potvrde interlock povratnog signala [s]. *)
	END_STRUCT;
	typParPGRad : 	STRUCT
		SetPritisakPotisa : REAL; (* Zadati pritisak potisa glavne pumpe [bar]. *)
		MinProtok : REAL; (* Donja granica protoka. *)
		MaxProtok : REAL; (* Gornja granica protoka. *)
		MinFR_Pumpe : REAL; (* Minimalni dozvoljeni protok izlazne pumpe [l/s]. *)
		MaxFR_Pumpe : REAL; (* Maksimalni dozvoljeni protok izlazne pumpe [l/s]. *)
		SetPointNivoTanka : REAL; (* Ciljani nivo prihvatnog tanka [m]. *)
		SetPointMinTempIspiranja : REAL; (* Minimalna temperatura za zavrsetak ispiranja [degC]. *)
		SetPointPritisakPV05Ispiranje : REAL; (* PT06 SP tokom preispiranja [bar]. *)
		SetPointPritisakUlazTanka : REAL; (* PT04 SP aktivnog ulaznog ventila [bar]. *)
		SetPointMaxPritisakDolaznaCev : REAL; (* PT06 SP cuvara instalacije [bar]. *)
		PocetnaFrekvencaIzlaznePumpe : REAL; (* PID tracking frekvenca pri startu [Hz]. *)
		MaxOtvorPropZaZatvaranje : REAL; (* Najveca otvorenost za potvrdu zatvaranja [%]. *)
		TimeSP : typTimeSPPGRad; (* RETAIN vremenski SP parametri u sekundama. *)
		AirRelease : typParAirReleasePGRad; (* RETAIN parametri PV03/PV04 za oba izvora. *)
	END_STRUCT;
	typCtrlAirReleasePGRad : 	STRUCT  (* HMI i servisne komande jednog odzracnog ventila. *)
		EnableManual : BOOL; (* TRUE = direktna rucna komanda ima prioritet nad automatikom. *)
		ManualSP_Percent : REAL; (* Direktna rucna komanda ventila [%]. *)
		ResetAlarm : BOOL; (* Pojedinacni jednokratni reset memorisanog alarma. *)
	END_STRUCT;
	typAirReleaseChannelPGRad : 	STRUCT  (* Izvrsni FB i komande jednog odzracnog ventila. *)
		FB : FB_AirRelease; (* Instanca upravljanja odzracivanjem. *)
		Ctrl : typCtrlAirReleasePGRad; (* HMI i servisne komande instance. *)
	END_STRUCT;
	typAirReleasePGRad : 	STRUCT  (* Grupisane runtime instance odzracivanja PV03/PV04. *)
		PV03 : typAirReleaseChannelPGRad; (* Odzracivanje ulaza u podstanicu. *)
		PV04 : typAirReleaseChannelPGRad; (* Odzracivanje ulaza u prihvatni tank. *)
	END_STRUCT;
	typCtrlPGRad : 	STRUCT
		SelektovaniIzvor : E_SelektovaniIzvor; (* Izbor izvora termalne vode. *)
		RegulacionaVarijanta : E_RegulacionaVarijanta; (* Izabrana regulaciona varijanta. *)
		AktivnaPumpaIzlazTanka : E_AktivnaPumpaIzlazTanka; (* Aktivna izlazna pumpa. *)
		AktivniPropVentilUlazTanka : E_AktivniPropVentilUlazTanka; (* Aktivni ulazni prop. ventil. *)
		AutoRestart : BOOL; (* Automatski start nakon cold boot-a. *)
	END_STRUCT;
	typManualPGRad : STRUCT
		Enable : BOOL; (* Dozvola servisnog rucnog rezima; aktivan samo u Standby. *)
		Sequence : USINT; (* Izabrana sekvenca: 1=BRB2 priprema/ispiranje, 2=IEBKB1 priprema, 3=kontrolisani stop. *)
		Start : BOOL; (* Impuls za pokretanje izabrane servisne sekvence. *)
		Stop : BOOL; (* Impuls za bezbedan prekid servisne sekvence. *)
		NextStep : BOOL; (* Impuls za zahtev sledeceg dozvoljenog podkoraka. *)
		Abort : BOOL; (* Impuls za povratak u Standby bez preskakanja stop logike. *)
	END_STRUCT;
	typCmdOnOffPGRad : 	STRUCT
		_03_Open : BOOL; (* PG_V03 - zahtev otvaranja izlazne grane pumpe 1. *)
		_04_Open : BOOL; (* PG_V04 - zahtev otvaranja izlazne grane pumpe 2. *)
		_05_Open : BOOL; (* PG_V05 - zahtev otvaranja bypass-a/preispiranja. *)
		_06_Open : BOOL; (* PG_V06 - zahtev otvaranja grane PV01 ka tanku. *)
		_07_Open : BOOL; (* PG_V07 - zahtev otvaranja grane PV02 ka tanku. *)
	END_STRUCT;
	typCmdPropVentilPGRad : 	STRUCT
		Enable : BOOL; (* Dozvola automatskog upravljanja ventilom. *)
		SP_Percent : REAL; (* Automatski zahtev otvorenosti 0..100%. *)
	END_STRUCT;
	typCmdPropVentiliPGRad : 	STRUCT
		PV01 : typCmdPropVentilPGRad; (* PG_PV01 - ulazni proporcionalni ventil 1. *)
		PV02 : typCmdPropVentilPGRad; (* PG_PV02 - ulazni proporcionalni ventil 2. *)
		PV05 : typCmdPropVentilPGRad; (* PG_PV05 - drenazni proporcionalni ventil. *)
	END_STRUCT;
	typCmdAirReleaseChannelPGRad : 	STRUCT  (* Procesna dozvola jednog odzracnog ventila. *)
		Enable : BOOL; (* TRUE = dozvoljen automatski ili rucni rad FB_AirRelease. *)
	END_STRUCT;
	typCmdAirReleasePGRad : 	STRUCT  (* Komandni vektor odzracivanja iz state masine. *)
		PV03 : typCmdAirReleaseChannelPGRad; (* Dozvola odzracivanja ulaza u podstanicu. *)
		PV04 : typCmdAirReleaseChannelPGRad; (* Dozvola odzracivanja ulaza u tank. *)
		UseIEBKB1Parameters : BOOL; (* TRUE = koristi IEBKB1, FALSE = koristi BRB2 parametre. *)
		ResetAll : BOOL; (* Zajednicki reset oba FB-a iz KomandaReset. *)
	END_STRUCT;
	typCmdPumpaPGRad : 	STRUCT
		Run : BOOL; (* Dozvola rada pumpe; frekvencu iskljucivo vodi PID_Pu_01. *)
	END_STRUCT;
	typCmdPumpePGRad : 	STRUCT
		_01 : typCmdPumpaPGRad; (* PG_Pu01 - komandni zahtev za izlaznu pumpu 1. *)
		_02 : typCmdPumpaPGRad; (* PG_Pu02 - komandni zahtev za izlaznu pumpu 2. *)
	END_STRUCT;
	typCmdPIDPumpePGRad : 	STRUCT
		Enable : BOOL; (* Dozvola rada jedinog PID_Pu_01 regulatora. *)
		ActValue : REAL; (* Aktivna regulisana vrednost: nivo tanka ili PT05 [m/bar]. *)
		SetValue : REAL; (* SP aktivne regulisane vrednosti [m/bar]. *)
		Invert : BOOL; (* Smer PID-a: TRUE za nivo, FALSE za pritisak. *)
		MaxOut : REAL; (* Maksimalni frekventni izlaz izabrane pumpe [Hz]. *)
		EnableTracking : BOOL; (* Dozvola bumpless starta na TrackingValue. *)
		TrackingValue : REAL; (* Pocetni frekventni zahtev PID-a pri startu [Hz]. *)
	END_STRUCT;
	typVezaPGRadBRB2 : 	STRUCT
		RadKaPodstanici : BOOL; (* PT izbor rute BRB2 ka podstanici; prihvata se samo u BRB2 standby. *)
		ManualMode : BOOL; (* Dozvola servisnog rucnog rezima. *)
		ManualSequence : USINT; (* Izabrana servisna sekvenca. *)
		ManualStart : BOOL; (* Impuls za pokretanje servisne sekvence. *)
		ManualStop : BOOL; (* Impuls za bezbedan prekid servisne sekvence. *)
		ManualNextStep : BOOL; (* Impuls za sledeci dozvoljeni podkorak. *)
		ManualAbort : BOOL; (* Impuls za povratak u Standby. *)
		ZahtevStarta : BOOL; (* PT zahtev BRB2 za pripremu i start bunarske pumpe. *)
		ZahtevZaustavljanja : BOOL; (* PT zahtev BRB2 za kontrolisano zaustavljanje. *)
		VentiliPodstaniceZatvoreni : BOOL; (* PT potvrda zatvorenosti PG_PV01, PG_PV02 i PG_PV05. *)
		PritisakIEBKB1 : REAL; (* PT prosledjuje stvarni pritisak IEBKB1 odredista [bar]. *)
		PodstanicaURezimuRada : BOOL; (* PT tank je na nivou i izabrana izlazna pumpa je stvarno u radu. *)
		PumpaAktivna : BOOL; (* BRB2 stvarna potvrda da je RB2_01 u InRun stanju. *)
		IspiranjeProtokDostignut : BOOL; (* BRB2 stvarni protok je dostigao ProtokIspiranja. *)
		IspiranjeMinTrajanjeDostignuto : BOOL; (* BRB2 je na ProtokIspiranja najmanje T_IspiranjeMin. *)
		StopSPDostignut : BOOL; (* BRB2 potvrda dostignutog FR_MinZeroFlow. *)
		RB2V01Zatvoren : BOOL; (* BRB2 potvrda zatvorenog RB2_V01 za IEBKB1 granu. *)
		RB2V02Zatvoren : BOOL; (* BRB2 potvrda zatvorenog RB2_V02. *)
	END_STRUCT;
	typCmdPGRad : 	STRUCT
		Aktivan : BOOL; (* State masina je vlasnik neretentivnih fizickih komandi. *)
		Ventili : typCmdOnOffPGRad; (* Zahtevi automatskih ON/OFF ventila. *)
		PropVentili : typCmdPropVentiliPGRad; (* Zahtevi proporcionalnih ventila. *)
		AirRelease : typCmdAirReleasePGRad; (* Zahtevi odzracivanja PV03/PV04. *)
		Pumpe : typCmdPumpePGRad; (* Zahtevi izlaznih pumpi. *)
		PID : typCmdPIDPumpePGRad; (* Ulazi jedinog PID-a izlazne pumpe. *)
	END_STRUCT;
	typPGRadStatus : 	STRUCT
		State : USINT; (* Eksplicitni PGRad state kod za komunikaciju i HMI. *)
		StateComment : STRING[80]; (* Operaterski opis aktivnog stanja. *)
		Substep : USINT; (* Aktivni podkorak state masine. *)
		SubstepComment : STRING[80]; (* Operaterski opis aktivnog podkoraka. *)
		Fault : BOOL; (* Zakacena procesna greska. *)
		FaultCode : USINT; (* Sifra zakacene procesne greske. *)
	END_STRUCT;
	typPGRadTrendCursor : 	STRUCT
		Position : REAL; (* Normalizovana pozicija kursora: 0.0 = levo, 1.0 = desno. *)
		Time : UDINT; (* Proteklo vreme od pocetka trend zapisa na poziciji kursora [ms]. *)
		RecordingStart : DATE_AND_TIME; (* Apsolutno vreme pocetka referentnog trend zapisa. *)
		DateTime : DATE_AND_TIME; (* Apsolutni datum i vreme uzorka na poziciji kursora. *)
		ViewStart : DATE_AND_TIME; (* Leva granica trenutno prikazanog vremenskog prozora. *)
		ViewSpan : DINT; (* Sirina prikazanog vremenskog prozora [s]. *)
		AxisMode : UINT; (* VC time-scale mod: 0 = zadati prozor bez automatskog pomeranja. *)
		PreviousViewSpan : DINT; (* Prethodna sirina prozora za promenu zoom-a bez skoka. *)
		FollowNow : BOOL; (* TRUE = desna ivica prozora prati trenutno vreme. *)
		CmdBack : BOOL; (* Jednokratni zahtev za prethodni vremenski prozor. *)
		CmdForward : BOOL; (* Jednokratni zahtev za sledeci vremenski prozor. *)
		CmdNow : BOOL; (* Jednokratni zahtev za povratak na najnovije podatke. *)
		AxisTime0 : DATE_AND_TIME; (* Pocetak prikazanog vremenskog prozora. *)
		AxisTime1 : DATE_AND_TIME; (* Prva unutrasnja vremenska oznaka ose. *)
		AxisTime2 : DATE_AND_TIME; (* Druga unutrasnja vremenska oznaka ose. *)
		AxisTime3 : DATE_AND_TIME; (* Treca unutrasnja vremenska oznaka ose. *)
		AxisTime4 : DATE_AND_TIME; (* Cetvrta unutrasnja vremenska oznaka ose. *)
		AxisTime5 : DATE_AND_TIME; (* Peta unutrasnja vremenska oznaka ose. *)
		AxisTime6 : DATE_AND_TIME; (* Sesta unutrasnja vremenska oznaka ose. *)
		AxisTime7 : DATE_AND_TIME; (* Sedma unutrasnja vremenska oznaka ose. *)
		AxisTime8 : DATE_AND_TIME; (* Kraj prikazanog vremenskog prozora. *)
		Status : UINT; (* VC status trend kursora; bit 10 oznacava validan Cursor 1. *)
		Nivo : REAL; (* Nivo prihvatnog tanka na poziciji kursora [m]. *)
		Pritisak : REAL; (* PT05 pritisak potisa pumpe na poziciji kursora [bar]. *)
		Protok : REAL; (* Protok ka bazenima na poziciji kursora [l/s]. *)
		TT01 : REAL; (* Temperatura TT01 na poziciji kursora [degC]. *)
		TT03 : REAL; (* Temperatura u prihvatnom tanku TT03 na poziciji kursora [degC]. *)
		TT04 : REAL; (* Temperatura TT04 na poziciji kursora [degC]. *)
		TT05 : REAL; (* Temperatura TT05 na poziciji kursora [degC]. *)
		TT06 : REAL; (* Temperatura TT06 na poziciji kursora [degC]. *)
	END_STRUCT;
	typPGRad : 	STRUCT
		CmdRetain : typCmdRetainUlazniVentiliPGRad; (* Retain komande bistabilnih ulaznih ventila. *)
		Par : typParPGRad; (* Retain projektni parametri procesa podstanice. *)
		Ctrl : typCtrlPGRad; (* Retain HMI izbor izvora i regulacije. *)
	END_STRUCT;
END_TYPE
```

### Global.var - Global variables
```iecst
VAR RETAIN
	(* Lokalni izbor automatskog rada izlazne pumpe. *)
	Pu_01_Auto : BOOL;
	PGRad : typPGRad; (* Retain procesni kontekst podstanice: Ctrl, Par i CmdRetain. *)
END_VAR

VAR
	(* Izracunate procesne vrednosti za HMI i nadzor. *)
	AktivniUlazniProtok : REAL; (* Realni protok aktivnog izvora termalne vode [l/s]. *)
	Predata_Snaga : REAL; (* Ukupna snaga predata izmenjivacima [kW]. *)
	Snaga_grejanja_hotela : REAL; (* Snaga predata hotelskom grejanju [kW]. *)
	Snaga_sanitarnog_grejanja : REAL; (* Preostala snaga predata sanitarnom grejanju [kW]. *)
	DP_Izmejnivac : REAL;
	DP_strainer : REAL;
	NivoPRihvatniSud : REAL;
	PG : PG_type; (* Korenski I/O i HMI objekat podstanice: Act i Sens bez retain-a. *)

	(* Lokalni PID izlazne pumpe. *)
	PID_Pu_01 : MTBasicsPID;
	startPIDPu1 : BOOL;

	(* Neretentivni PT komandni vektor i PT-BRB2 komunikacioni ugovor. *)
	PGRad_Cmd : typCmdPGRad; (* Neretentivni vektor: Rad_PG_KB pise, PID i IO ga primenjuju. *)
	PGRad_BRB2Cmd : typVezaPGRadBRB2; (* Kanonski PT izlazni status; pise samo Rad_PG_KB. *)
	PGRad_BRB2 : typVezaPGRadBRB2; (* Lokalni procesni ugovor; pise samo PG_Intf. *)
	PGRad_BRB2_Tx : typVezaPGRadBRB2; (* PT izlazni AsIMA snapshot; pise samo PG_Intf. *)
	PGRad_BRB2_Rx : typVezaPGRadBRB2; (* BRB2 ulazni AsIMA snapshot; pise samo IMAcomm. *)
	PGRad_Status : typPGRadStatus; (* Process status DTO za HMI i AsIMA snapshot. *)
	PGRad_AirRelease : typAirReleasePGRad; (* Runtime FB instance i HMI komande odzracivanja PV03/PV04. *)
	PGRad_TrendCursor : typPGRadTrendCursor; (* Vreme i procesne vrednosti na poziciji HMI trend kursora. *)
END_VAR
```

### PG01.typ - PG01 AsIMA synoptic data types
```iecst
TYPE
	typPG01SynVentil : 	STRUCT  (* Sinopticki komandni i statusni podaci jednog ON/OFF ventila. *)
		OpenCmd : BOOL; (* Lokalna komanda otvaranja. *)
		CloseCmd : BOOL; (* Lokalna komanda zatvaranja. *)
		Opened : BOOL; (* Povratni signal otvorenog polozaja. *)
		Closed : BOOL; (* Povratni signal zatvorenog polozaja. *)
		Alarm : BOOL; (* Dijagnosticki alarm ventila. *)
	END_STRUCT;
	typPG01SynPropVentil : 	STRUCT  (* Sinopticki komandni i statusni podaci jednog proporcionalnog ventila. *)
		Enable : BOOL; (* Dozvola automatske regulacije. *)
		CmdPercent : REAL; (* Zadata otvorenost [%]. *)
		PositionPercent : REAL; (* Ostvarena otvorenost [%]. *)
		Alarm : BOOL; (* Dijagnosticki alarm ventila. *)
	END_STRUCT;
	typPG01SynPumpa : 	STRUCT  (* Sinopticki komandni i statusni podaci jedne pumpe. *)
		RunCmd : BOOL; (* Lokalni zahtev rada. *)
		Running : BOOL; (* Stvarni status rada. *)
		Frequency : REAL; (* Frekventni zahtev/ostvarenje [Hz]. *)
		Alarm : BOOL; (* Dijagnosticki alarm pumpe. *)
	END_STRUCT;
	typPG01SynAnalog : 	STRUCT  (* Sinopticki podatak jednog analognog procesnog signala. *)
		Value : REAL; (* Skalirana merena vrednost. *)
		Valid : BOOL; (* Validnost signala. *)
		Alarm : BOOL; (* Dijagnosticki alarm signala. *)
	END_STRUCT;
	typPG01SynDigital : 	STRUCT  (* Sinopticki podatak jednog digitalnog procesnog signala. *)
		Value : BOOL; (* Digitalna merena vrednost. *)
		Alarm : BOOL; (* Dijagnosticki alarm signala. *)
	END_STRUCT;
	typPG01SynPGAct : 	STRUCT  (* Lokalni PT aktuatori koje Podstanica objavljuje BRB2-u i sinoptici. *)
		Pu01 : typPG01SynPumpa; (* PG_Pu01 - prva izlazna pumpa prihvatnog tanka. *)
		Pu02 : typPG01SynPumpa; (* PG_Pu02 - druga izlazna pumpa prihvatnog tanka. *)
		PV01 : typPG01SynPropVentil; (* PG_PV01 - prvi regulacioni ulaz u tank. *)
		PV02 : typPG01SynPropVentil; (* PG_PV02 - drugi regulacioni ulaz u tank. *)
		PV03 : typPG01SynPropVentil; (* PG_PV03 - odzracni proporcionalni ventil na ulazu u Podstanicu. *)
		PV04 : typPG01SynPropVentil; (* PG_PV04 - odzracni proporcionalni ventil na ulazu u tank. *)
		PV05 : typPG01SynPropVentil; (* PG_PV05 - regulacioni/drenazni ventil BRB2 grane. *)
		AV01 : typPG01SynVentil; (* PG_AV01 - lokalni automatski ventil; funkcija se vidi iz PT procesne logike. *)
		AV02 : typPG01SynVentil; (* PG_AV02 - lokalni automatski ventil; funkcija se vidi iz PT procesne logike. *)
		AV03 : typPG01SynVentil; (* PG_AV03 - izlazna grana pumpe PG_Pu01. *)
		AV04 : typPG01SynVentil; (* PG_AV04 - izlazna grana pumpe PG_Pu02. *)
		AV05 : typPG01SynVentil; (* PG_AV05 - bypass/preispiranje Podstanice. *)
		AV06 : typPG01SynVentil; (* PG_AV06 - grana PG_PV01 ka prihvatnom tanku. *)
		AV07 : typPG01SynVentil; (* PG_AV07 - grana PG_PV02 ka prihvatnom tanku. *)
		RV19 : typPG01SynVentil; (* PG_RV19 - rucni ventil posle PG_PV01. *)
		RV21 : typPG01SynVentil; (* PG_RV21 - rucni ventil posle PG_PV02. *)
		RV22 : typPG01SynVentil; (* PG_RV22 - drenazni ventil na dnu prihvatnog tanka. *)
		RV23 : typPG01SynVentil; (* PG_RV23 - ulazni rucni ventil pumpe PG_Pu01. *)
		RV24 : typPG01SynVentil; (* PG_RV24 - ulazni rucni ventil pumpe PG_Pu02. *)
		RV25 : typPG01SynVentil; (* PG_RV25 - bypassni izlaz gasa iz prihvatnog tanka. *)
		RV26 : typPG01SynVentil; (* PG_RV26 - ulazni rucni ventil vakuum pumpe. *)
		RV27 : typPG01SynVentil; (* PG_RV27 - izlazni rucni ventil vakuum pumpe. *)
	END_STRUCT;
	typPG01SynPGSens : 	STRUCT  (* Lokalni PT senzorski snapshot; analogne vrednosti koriste procesne jedinice. *)
		Pt00 : typPG01SynAnalog; (* Pritisak komprimovanog vazduha [bar]. *)
		Pt01 : typPG01SynAnalog; (* Pritisak termalne vode na ulazu u Podstanicu [bar]. *)
		Pt02 : typPG01SynAnalog; (* PT_PG_02 - pritisak posle grubih filtera [bar]. *)
		Pt03 : typPG01SynAnalog; (* PT_PG_03 - pritisak posle velikog izmenjivaca [bar]. *)
		Pt04 : typPG01SynAnalog; (* PT_PG_04 - pritisak na ulazu u prihvatni tank [bar]. *)
		Pt05 : typPG01SynAnalog; (* PT_PG_05 - pritisak na potisu izlaznih pumpi [bar]. *)
		Pt06 : typPG01SynAnalog; (* PT_PG_06 - pritisak BRB2 magistrale pre PG_V02 [bar]. *)
		PtNS1 : typPG01SynAnalog; (* Pritisak na dnu prihvatnog tanka [mbar]. *)
		PtNS2 : typPG01SynAnalog; (* Pritisak na vrhu prihvatnog tanka [mbar]. *)
		Tt01 : typPG01SynAnalog; (* TT_PG_01 - ulaz u veliki izmenjivac [degC]. *)
		Tt02 : typPG01SynAnalog; (* TT_PG_02 - ulaz u prihvatni tank [degC]. *)
		Tt03 : typPG01SynAnalog; (* TT_PG_03 - temperatura prihvatnog tanka [degC]. *)
		Tt04 : typPG01SynAnalog; (* TT_PG_04 - izlaz iz velikog izmenjivaca [degC]. *)
		Tt05 : typPG01SynAnalog; (* TT_PG_05 - ulaz u mali izmenjivac [degC]. *)
		Tt06 : typPG01SynAnalog; (* TT_PG_06 - izlaz iz malog izmenjivaca [degC]. *)
		Tt07 : typPG01SynAnalog; (* TT_PG_07 - drenazni vod za potvrdu preispiranja [degC]. *)
		Tt08 : typPG01SynAnalog; (* TT_PG_08 - ulaz tehnicke vode u direktni izmenjivac. *)
		Tt09 : typPG01SynAnalog; (* TT_PG_09 - izlaz tehnicke vode iz direktnog izmenjivaca. *)
		Tt10 : typPG01SynAnalog; (* TT_PG_10 - ulaz sanitarne vode u direktni izmenjivac. *)
		Tt11 : typPG01SynAnalog; (* TT_PG_11 - izlaz sanitarne vode iz direktnog izmenjivaca. *)
		MP01 : typPG01SynAnalog; (* MP_PG_01 - protok ka potrosacima [m3/h]. *)
		LS01 : typPG01SynDigital; (* LS_PG_01 - nizak nivo prihvatnog tanka. *)
		LS02 : typPG01SynDigital; (* LS_PG_02 - donji nivo prvog odzracnog cilindra. *)
		LS03 : typPG01SynDigital; (* LS_PG_03 - gornji nivo prvog odzracnog cilindra. *)
		LS04 : typPG01SynDigital; (* LS_PG_04 - donji nivo drugog odzracnog cilindra. *)
		LS05 : typPG01SynDigital; (* LS_PG_05 - gornji nivo drugog odzracnog cilindra. *)
		OWF01 : typPG01SynDigital; (* PG_OWF01 - status prvog zastitnog prestrujnog ventila. *)
		OWF02 : typPG01SynDigital; (* PG_OWF02 - status drugog zastitnog prestrujnog ventila. *)
	END_STRUCT;
	typPG01SynPGCtrl : 	STRUCT  (* Lokalni PT izbori, stanje i procesna dijagnostika za sinoptiku. *)
		Izvor : USINT; (* E_SelektovaniIzvor kao numericka vrednost. *)
		Regulacija : USINT; (* E_RegulacionaVarijanta kao numericka vrednost. *)
		IzlaznaPumpa : USINT; (* E_AktivnaPumpaIzlazTanka kao numericka vrednost. *)
		UlazniPV : USINT; (* E_AktivniPropVentilUlazTanka kao numericka vrednost. *)
		AutoRestart : BOOL; (* RETAIN zahtev automatskog ponovnog pokretanja nakon cold boot-a. *)
		State : USINT; (* E_PGRad_State kao numericka vrednost. *)
		Substep : USINT; (* Aktivni podkorak unutar glavnog procesnog stanja. *)
		Fault : BOOL; (* Zbirni procesni fault Podstanice. *)
		FaultCode : USINT; (* Numericka sifra uzroka procesnog fault-a. *)
	END_STRUCT;
	typPG01SynBRB2Act : 	STRUCT  (* Udaljeni BRB2 aktuatori koje BRB2 pise, a Podstanica samo prikazuje. *)
		RB101 : typPG01SynPumpa; (* BRB2 pumpa oznake RB1_01; udaljeni status/komanda. *)
		RB201 : typPG01SynPumpa; (* BRB2 pumpa oznake RB2_01; udaljeni status/komanda. *)
		RB202 : typPG01SynPumpa; (* BRB2 pumpa oznake RB2_02; udaljeni status/komanda. *)
		RB211 : typPG01SynPumpa; (* BRB2 pumpa oznake RB2_11; udaljeni status/komanda. *)
		AVRB1V01 : typPG01SynVentil; (* BRB2 automatski ventil RB1_V01; udaljeni status/komanda. *)
		AVRB1V02 : typPG01SynVentil; (* BRB2 automatski ventil RB1_V02; udaljeni status/komanda. *)
		AVRB2V01 : typPG01SynVentil; (* BRB2 automatski ventil RB2_V01; udaljeni status/komanda. *)
		AVRB2V02 : typPG01SynVentil; (* BRB2 automatski ventil RB2_V02; udaljeni status/komanda. *)
		AVRB2V20 : typPG01SynVentil; (* BRB2 automatski ventil RB2_V20; udaljeni status/komanda. *)
		AVRB2V21 : typPG01SynVentil; (* BRB2 automatski ventil RB2_V21; udaljeni status/komanda. *)
		RVRB1RV04 : typPG01SynVentil; (* BRB2 rucni ventil RB1_RV04; udaljeni status. *)
		RVRB1RV05 : typPG01SynVentil; (* BRB2 rucni ventil RB1_RV05; udaljeni status. *)
		RVRB2RV04 : typPG01SynVentil; (* BRB2 rucni ventil RB2_RV04; udaljeni status. *)
		RVRB2RV05 : typPG01SynVentil; (* BRB2 rucni ventil RB2_RV05; udaljeni status. *)
		RVRB2RV06 : typPG01SynVentil; (* BRB2 rucni ventil RB2_RV06; udaljeni status. *)
		RVRB2RV10 : typPG01SynVentil; (* BRB2 rucni ventil RB2_RV10; udaljeni status. *)
		RVRB2RV51 : typPG01SynVentil; (* BRB2 rucni ventil RB2_RV51; udaljeni status. *)
		PVRB1PV01 : typPG01SynPropVentil; (* BRB2 proporcionalni ventil RB1_PV01; udaljeni status/komanda. *)
		PVRB2PV01 : typPG01SynPropVentil; (* BRB2 proporcionalni ventil RB2_PV01; udaljeni status/komanda. *)
		PVRB2PV11 : typPG01SynPropVentil; (* BRB2 proporcionalni ventil RB2_PV11; udaljeni status/komanda. *)
		PVRB2PV21 : typPG01SynPropVentil; (* BRB2 proporcionalni ventil RB2_PV21; udaljeni status/komanda. *)
	END_STRUCT;
	typPG01SynBRB2Sens : 	STRUCT  (* Udaljeni BRB2 senzori; vrednosti ostaju u jedinicama izvornog PLC-a. *)
		PtAir : typPG01SynAnalog; (* BRB2 pritisak vazduha; jedinica i fizicki identitet nepotvrdjeni u PT kodu. *)
		PtColdWater : typPG01SynAnalog; (* BRB2 pritisak hladne vode; jedinica i fizicki identitet nepotvrdjeni u PT kodu. *)
		PtRB10 : typPG01SynAnalog; (* BRB2 senzor pritiska oznake RB10; jedinica prema udaljenom PLC-u. *)
		PtRB11 : typPG01SynAnalog; (* BRB2 senzor pritiska oznake RB11; jedinica prema udaljenom PLC-u. *)
		PtRB20A : typPG01SynAnalog; (* BRB2 senzor pritiska oznake RB20A; jedinica prema udaljenom PLC-u. *)
		PtRB20B : typPG01SynAnalog; (* BRB2 senzor pritiska oznake RB20B; jedinica prema udaljenom PLC-u. *)
		PtRB21 : typPG01SynAnalog; (* BRB2 senzor pritiska oznake RB21; jedinica prema udaljenom PLC-u. *)
		PtRB22 : typPG01SynAnalog; (* BRB2 senzor pritiska oznake RB22; jedinica prema udaljenom PLC-u. *)
		PtRB211 : typPG01SynAnalog; (* BRB2 senzor pritiska oznake RB211; jedinica prema udaljenom PLC-u. *)
		PtRB212 : typPG01SynAnalog; (* BRB2 senzor pritiska oznake RB212; jedinica prema udaljenom PLC-u. *)
		PtRB213 : typPG01SynAnalog; (* BRB2 senzor pritiska oznake RB213; jedinica prema udaljenom PLC-u. *)
		TtRB11 : typPG01SynAnalog; (* BRB2 senzor temperature oznake RB11; jedinica prema udaljenom PLC-u. *)
		TtRB21 : typPG01SynAnalog; (* BRB2 senzor temperature oznake RB21; jedinica prema udaljenom PLC-u. *)
		TtRB22 : typPG01SynAnalog; (* BRB2 senzor temperature oznake RB22; jedinica prema udaljenom PLC-u. *)
		TtRB211 : typPG01SynAnalog; (* BRB2 senzor temperature oznake RB211; jedinica prema udaljenom PLC-u. *)
		TtPump : typPG01SynAnalog; (* BRB2 temperatura pumpe; fizicki identitet nepotvrdjen u PT kodu. *)
		FtRB11 : typPG01SynAnalog; (* BRB2 senzor protoka oznake RB11; jedinica prema udaljenom PLC-u. *)
		FtRB21 : typPG01SynAnalog; (* BRB2 senzor protoka oznake RB21; jedinica prema udaljenom PLC-u. *)
		FtRB211 : typPG01SynAnalog; (* BRB2 senzor protoka oznake RB211; jedinica prema udaljenom PLC-u. *)
		KRB211 : typPG01SynAnalog; (* BRB2 senzor provodnosti oznake RB211; jedinica prema udaljenom PLC-u. *)
		RHT01T : typPG01SynAnalog; (* BRB2 temperatura senzora RHT01; jedinica prema udaljenom PLC-u. *)
		RHT01RH : typPG01SynAnalog; (* BRB2 relativna vlaznost senzora RHT01; jedinica prema udaljenom PLC-u. *)
		RHT02T : typPG01SynAnalog; (* BRB2 temperatura senzora RHT02; jedinica prema udaljenom PLC-u. *)
		RHT02RH : typPG01SynAnalog; (* BRB2 relativna vlaznost senzora RHT02; jedinica prema udaljenom PLC-u. *)
		RHT03T : typPG01SynAnalog; (* BRB2 temperatura senzora RHT03; jedinica prema udaljenom PLC-u. *)
		RHT03RH : typPG01SynAnalog; (* BRB2 relativna vlaznost senzora RHT03; jedinica prema udaljenom PLC-u. *)
		LSRB11 : typPG01SynDigital; (* BRB2 binarni nivo signal oznake RB11; fizicki identitet nepotvrdjen. *)
		LSRB21 : typPG01SynDigital; (* BRB2 binarni nivo signal oznake RB21; fizicki identitet nepotvrdjen. *)
		OWFRB101 : typPG01SynDigital; (* BRB2 prestrujni zastitni signal oznake RB101. *)
		OWFRB201 : typPG01SynDigital; (* BRB2 prestrujni zastitni signal oznake RB201. *)
		OWFRB202 : typPG01SynDigital; (* BRB2 prestrujni zastitni signal oznake RB202. *)
	END_STRUCT;
	typPG01SynBRB2Ctrl : 	STRUCT  (* Udaljeni BRB2 procesni izbori, stanje i potvrde za PT sinoptiku. *)
		Odrediste : USINT; (* E_OdredisteBRB2 kao numericka vrednost. *)
		Regulacija : USINT; (* E_RegulacionaVarijanta kao numericka vrednost. *)
		Ispiranje : BOOL; (* BRB2 potvrda da je aktivna faza ispiranja/punjenja cevovoda. *)
		Aktivan : BOOL; (* BRB2 state masina trenutno poseduje fizicke komande. *)
		StopFaza : USINT; (* E_FazaZaustavljanjaBRB2 kao numericka vrednost. *)
		PumpaPotvrdjena : BOOL; (* BRB2 potvrda stvarnog rada aktivne pumpe. *)
		StopSPDostignut : BOOL; (* BRB2 potvrda dostignute minimalne frekvencije pri stopu. *)
		RB2V02Zatvoren : BOOL; (* BRB2 potvrda zatvorenog ventila RB2_V02. *)
	END_STRUCT;
	typPG01Syn : 	STRUCT  (* Zbirni PT/BRB2 snapshot za razmenu i prikaz na sinoptici. *)
		PGAct : typPG01SynPGAct; (* PT Act snapshot za sinoptiku. *)
		PGSens : typPG01SynPGSens; (* PT Sens snapshot za sinoptiku. *)
		PGCtrl : typPG01SynPGCtrl; (* PT Ctrl i state snapshot. *)
		BRB2Act : typPG01SynBRB2Act; (* BRB2 Act snapshot za sinoptiku. *)
		BRB2Sens : typPG01SynBRB2Sens; (* BRB2 Sens snapshot za sinoptiku. *)
		BRB2Ctrl : typPG01SynBRB2Ctrl; (* BRB2 Ctrl i state snapshot. *)
	END_STRUCT;
END_TYPE
```

### PG01.var - PG01 AsIMA synoptic variables
```iecst
VAR
	(* PT publish vektor: PT Act, Sens i Ctrl podatke salje prema BRB2/HMI. *)
	PG01_Local : typPG01Syn; (* PT upisuje lokalni Act/Sens/Ctrl snapshot za BRB2 i HMI. *)

	(* BRB2 mirror vektor: prima se samo za sinoptiku i ne upravlja PT opremom. *)
	PG01_Remote : typPG01Syn; (* BRB2 upisuje udaljeni snapshot; PT ga koristi samo za prikaz. *)
END_VAR
```

### IEB_KB1_Comm.typ - IEBKB1 remote mirror data types
```iecst
TYPE
	(* Sirova i skalirana referenca/povratna vrednost proporcionalnog ventila. *)
	ST_VALVE_PV_ACT : STRUCT (* Sirova i skalirana referenca/povratna vrednost proporcionalnog ventila. *)
		iREF_RAW : INT; (* Sirova referentna vrednost izlaza. *)
		rREF : REAL; (* Skalirana referentna vrednost. *)
		iFB_RAW : INT; (* Sirova povratna vrednost polozaja. *)
		rFB_SCALED : REAL; (* Skalirani povratni polozaj ventila. *)
	END_STRUCT;
	(* Status, komande, vremena i izbor rezima automatskog ventila. *)
	ST_VALVE_ACT_TYPE : STRUCT (* Status, komande, vremena i izbor rezima automatskog ventila. *)
		iSTATUS : INT; (* Kod radnog statusa ventila. *)
		xOPEN_FB : BOOL; (* Povratna potvrda otvorenog polozaja. *)
		xCLOSE_FB : BOOL; (* Povratna potvrda zatvorenog polozaja. *)
		xREQUEST : BOOL; (* Zahtev za promenu polozaja ventila. *)
		xSET : BOOL; (* Zadata binarna komanda polozaja. *)
		xVALVE_ALARM : BOOL; (* Zbirni alarm ventila. *)
		xAlarm_RESET : BOOL; (* Zahtev za reset alarma ventila. *)
		iCounter_Act : UDINT; (* Brojac aktivacija ventila. *)
		xCounter_RESET : BOOL; (* Zahtev za reset brojaca aktivacija. *)
		T_MAX_Preclosing_ms : UDINT; (* Maksimalni timeout predzatvaranja [ms]. *)
		T_MIN_Closing_ms : UDINT; (* Minimalno vreme zatvaranja [ms]. *)
		T_MAX_Closing_ms : UDINT; (* Maksimalni timeout zatvaranja [ms]. *)
		T_MAX_Preopening_ms : UDINT; (* Maksimalni timeout predotvaranja [ms]. *)
		T_MIN_Opening_ms : UDINT; (* Minimalno vreme otvaranja [ms]. *)
		T_MAX_Opening_ms : UDINT; (* Maksimalni timeout otvaranja [ms]. *)
		T_Preopening_ms : UDINT; (* Izmereno vreme predotvaranja [ms]. *)
		T_Opening_ms : UDINT; (* Izmereno vreme otvaranja [ms]. *)
		T_Preclosing_ms : UDINT; (* Izmereno vreme predzatvaranja [ms]. *)
		T_Closing_ms : UDINT; (* Izmereno vreme zatvaranja [ms]. *)
		xMANUAL_SET : BOOL; (* Rucna komanda polozaja. *)
		xMODE_AUTO_MAN : BOOL; (* Izbor automatskog ili rucnog rezima. *)
	END_STRUCT;
	(* Osnovni udaljeni analogni senzor; IEBKB1 upisuje merenje i status. *)
	ST_SENSORS_TYPE : STRUCT (* Osnovni udaljeni analogni senzor; IEBKB1 upisuje merenje i status. *)
		_00_raw_value : INT; (* Sirova vrednost senzora. *)
		_01_value : REAL; (* Skalirana procesna vrednost. *)
		_02_status : BOOL; (* Validnost/status senzora. *)
	END_STRUCT;
	(* Prosireni udaljeni analogni senzor sa dva dodatna binarna statusa. *)
	ST_SENSORS_K_TYPE : STRUCT (* Prosireni udaljeni analogni senzor sa dva dodatna binarna statusa. *)
		_00_raw_value : INT; (* Sirova vrednost senzora. *)
		_01_value : REAL; (* Skalirana procesna vrednost. *)
		_02_status : BOOL; (* Validnost/status senzora. *)
		_03_CB_1 : BOOL; (* Dodatni binarni status CB_1. *)
		_04_CB_2 : BOOL; (* Dodatni binarni status CB_2. *)
	END_STRUCT;
	(* Udaljeni status i komande pumpe/frekventnog regulatora. *)
	ST_PUMP : STRUCT (* Udaljeni status i komande pumpe/frekventnog regulatora. *)
		x_RUN : BOOL; (* Status rada pumpe. *)
		xAL : BOOL; (* Alarm pumpe ili regulatora. *)
		xAL_RST : BOOL; (* Zahtev za reset alarma. *)
		rFR_REF_scaled : REAL; (* Skalirana referenca frekvencije [Hz]. *)
		iFR_REF_raw : INT; (* Sirova referenca frekvencije. *)
	END_STRUCT;
	(* Udaljeni status rucnog ventila sa alarmnim vremenima. *)
	ST_MAN_VALVE : STRUCT (* Udaljeni status rucnog ventila sa alarmnim vremenima. *)
		xCLOSE_FB : BOOL; (* Povratna potvrda zatvorenog polozaja. *)
		xOPEN_FB : BOOL; (* Povratna potvrda otvorenog polozaja. *)
		xALARM_RESET : BOOL; (* Zahtev za reset alarma. *)
		rALARM_DELAY_PT : REAL; (* Zadato kasnjenje alarma. *)
		rALARM_ET : REAL; (* Proteklo vreme alarmnog uslova. *)
		xALARM : BOOL; (* Zbirni alarm ventila. *)
		iSTATUS : INT; (* Kod radnog statusa ventila. *)
	END_STRUCT;
	(* Udaljeni temperaturni senzori; IEBKB1 upisuje sve vrednosti/status. *)
	Sens_Tt_type : STRUCT (* Udaljeni temperaturni senzori; IEBKB1 upisuje sve vrednosti/status. *)
		B_00 : ST_SENSORS_TYPE; (* Uredjaj/signal oznake B_00 [degC]. *)
		B_01 : ST_SENSORS_TYPE; (* Uredjaj/signal oznake B_01 [degC]. *)
		B_02 : ST_SENSORS_TYPE; (* Uredjaj/signal oznake B_02 [degC]. *)
		B_101 : ST_SENSORS_TYPE; (* Uredjaj/signal oznake B_101 [degC]. *)
		B_111 : ST_SENSORS_TYPE; (* Uredjaj/signal oznake B_111 [degC]. *)
		B_201 : ST_SENSORS_TYPE; (* Uredjaj/signal oznake B_201 [degC]. *)
	END_STRUCT;
	(* Udaljeni senzori pritiska; IEBKB1 upisuje sve vrednosti/status. *)
	Sens_Pt_type : STRUCT (* Udaljeni senzori pritiska; IEBKB1 upisuje sve vrednosti/status. *)
		B_00 : ST_SENSORS_TYPE; (* Uredjaj/signal oznake B_00 [bar]. *)
		B_01 : ST_SENSORS_TYPE; (* Uredjaj/signal oznake B_01 [bar]. *)
		B_02 : ST_SENSORS_TYPE; (* Uredjaj/signal oznake B_02 [bar]. *)
		B_101 : ST_SENSORS_TYPE; (* Uredjaj/signal oznake B_101 [bar]. *)
		B_102 : ST_SENSORS_TYPE; (* Uredjaj/signal oznake B_102 [bar]. *)
		B_103 : ST_SENSORS_TYPE; (* Uredjaj/signal oznake B_103 [bar]. *)
		B_111 : ST_SENSORS_TYPE; (* Uredjaj/signal oznake B_111 [bar]. *)
		B_112 : ST_SENSORS_TYPE; (* Uredjaj/signal oznake B_112 [bar]. *)
		B_113 : ST_SENSORS_TYPE; (* Uredjaj/signal oznake B_113 [bar]. *)
		B_140 : ST_SENSORS_TYPE; (* Uredjaj/signal oznake B_140 [bar]. *)
		B_200 : ST_SENSORS_TYPE; (* Uredjaj/signal oznake B_200 [bar]. *)
		B_201 : ST_SENSORS_TYPE; (* Uredjaj/signal oznake B_201 [bar]. *)
		B_521 : ST_SENSORS_TYPE; (* Uredjaj/signal oznake B_521 [bar]. *)
	END_STRUCT;
	(* Udaljeni statusi napajanja; IEBKB1 upisuje stanje osiguraca i izvora. *)
	Sens_Power_type : STRUCT (* Udaljeni statusi napajanja; IEBKB1 upisuje stanje osiguraca i izvora. *)
		Fuse_DC : BOOL; (* Status DC osiguraca. *)
		Fuse_AC : BOOL; (* Status AC osiguraca. *)
		Suply_24VDC_1 : BOOL; (* Status prvog 24 VDC napajanja. *)
		Suply_24VDC_2 : BOOL; (* Status drugog 24 VDC napajanja. *)
		DC_UPS_1 : BOOL; (* Status prvog DC UPS izvora. *)
		DC_UPS_2 : BOOL; (* Status drugog DC UPS izvora. *)
	END_STRUCT;
	(* Udaljeno pH merenje; IEBKB1 upisuje vrednost i status. *)
	Sens_pH_type : STRUCT (* Udaljeno pH merenje; IEBKB1 upisuje vrednost i status. *)
		proba : ST_SENSORS_TYPE; (* pH sonda. *)
	END_STRUCT;
	(* Udaljeni meraci protoka; IEBKB1 upisuje vrednosti i status. *)
	Sens_MP_type : STRUCT (* Udaljeni meraci protoka; IEBKB1 upisuje vrednosti i status. *)
		B_01 : ST_SENSORS_TYPE; (* Uredjaj/signal oznake B_01 [protok]. *)
		B_02 : ST_SENSORS_TYPE; (* Uredjaj/signal oznake B_02 [protok]. *)
	END_STRUCT;
	(* Udaljeni binarni senzori nivoa; IEBKB1 upisuje stanja. *)
	Sens_LS_type : STRUCT (* Udaljeni binarni senzori nivoa; IEBKB1 upisuje stanja. *)
		B_01 : BOOL; (* Uredjaj/signal oznake B_01. *)
		B_101 : BOOL; (* Uredjaj/signal oznake B_101. *)
		B_102 : BOOL; (* Uredjaj/signal oznake B_102. *)
		B_111 : BOOL; (* Uredjaj/signal oznake B_111. *)
		B_112 : BOOL; (* Uredjaj/signal oznake B_112. *)
		B_201 : BOOL; (* Uredjaj/signal oznake B_201. *)
		B_301 : BOOL; (* Uredjaj/signal oznake B_301. *)
	END_STRUCT;
	(* Udaljeno merenje provodnosti/kvaliteta; IEBKB1 upisuje vrednost i status. *)
	Sens_K_type : STRUCT (* Udaljeno merenje provodnosti/kvaliteta; IEBKB1 upisuje vrednost i status. *)
		proba : ST_SENSORS_TYPE; (* Merna sonda K. *)
	END_STRUCT;
	(* Zbirna struktura udaljenih IEBKB1 senzora. *)
	Sens_type : STRUCT (* Zbirna struktura udaljenih IEBKB1 senzora. *)
		Pt : Sens_Pt_type; (* Senzori pritiska. *)
		Tt : Sens_Tt_type; (* Senzori temperature. *)
		LS : Sens_LS_type; (* Binarni senzori nivoa. *)
		MP : Sens_MP_type; (* Meraci protoka. *)
		K : Sens_K_type; (* Merna sonda K. *)
		pH : Sens_pH_type; (* pH sonda. *)
		Power : Sens_Power_type; (* Statusi napajanja. *)
	END_STRUCT;
	(* Komunikacioni ugovor podstanice: PT pise Zahtev, IEBKB1 pise Status. *)
	Cntrl_Comm_Podstanica_type : STRUCT (* Komunikacioni ugovor: PT pise Zahtev, IEBKB1 pise Status. *)
		Zahtev : typPodstanicaZahtev; (* PT upisuje zahtev udaljenom IEBKB1. *)
		Parametri : typPodstanicaParametri; (* Dogovoreni radni parametri komunikacije. *)
		Status : typPodstanicaStatus; (* Udaljeni IEBKB1 upisuje procesni status. *)
	END_STRUCT;
	(* Zahtev koji PT upisuje udaljenom IEBKB1 sistemu. *)
	typPodstanicaZahtev : STRUCT (* Zahtev koji PT upisuje udaljenom IEBKB1 sistemu. *)
		ZahtevVode : BOOL; (* PT zahtev za dotok vode. *)
		NivoPrihvatnogTanka : REAL; (* PT izmereni nivo prihvatnog tanka [m]. *)
		CiljaniProtok : REAL; (* PT zadati ciljani protok. *)
		ModRada : USINT; (* PT zadati kod rezima rada. *)
	END_STRUCT;
	(* Granice protoka i frekvencije razmenjene sa udaljenim IEBKB1. *)
	typPodstanicaParametri : STRUCT (* Granice protoka i frekvencije razmenjene sa udaljenim IEBKB1. *)
		MinimalniProtok : REAL; (* Donja radna granica protoka. *)
		MaksimalniProtok : REAL; (* Gornja radna granica protoka. *)
		MinimalnaFrekvenca : REAL; (* Donja granica frekvencije [Hz]. *)
		MaksimalnaFrekvenca : REAL; (* Gornja granica frekvencije [Hz]. *)
		TolerancijaFrekvence : REAL; (* Dozvoljeno odstupanje frekvencije [Hz]. *)
	END_STRUCT;
	(* Procesni status koji udaljeni IEBKB1 upisuje PT sistemu. *)
	typPodstanicaStatus : STRUCT (* Procesni status koji udaljeni IEBKB1 upisuje PT sistemu. *)
		TrenutniProtok : REAL; (* Udaljeno izmereni trenutni protok. *)
		TrenutnaFrekvencaPumpe : REAL; (* Udaljena frekvencija pumpe [Hz]. *)
		MinimalniProtokDostignut : BOOL; (* Status dostignute minimalne granice protoka. *)
		MaksimalniProtokDostignut : BOOL; (* Status dostignute maksimalne granice protoka. *)
	END_STRUCT;
	(* Rezervisani komunikacioni prostor za BRB2. *)
	Cntrl_Comm_BRB2_type : STRUCT (* Rezervisani komunikacioni prostor za BRB2. *)
		Reserved : USINT; (* Rezervisano za buduce prosirenje ugovora. *)
	END_STRUCT;
	(* Zbirni komunikacioni ugovor upravljanja. *)
	Cntrl_Comm_type : STRUCT (* Zbirni komunikacioni ugovor upravljanja. *)
		Podstanica : Cntrl_Comm_Podstanica_type; (* Ugovor PT podstanice i IEBKB1. *)
		BRB2 : Cntrl_Comm_BRB2_type; (* Rezervisani BRB2 komunikacioni deo. *)
	END_STRUCT;
	(* Zbirni kontrolni podaci komunikacije IEBKB1. *)
	Cntrl_type : STRUCT (* Zbirni kontrolni podaci komunikacije IEBKB1. *)
		proba : BOOL; (* Pomocni komunikacioni/kontrolni signal. *)
		State : INT; (* Kod trenutnog kontrolnog stanja. *)
		Comm : Cntrl_Comm_type; (* Strukturirani komunikacioni ugovor. *)
	END_STRUCT;
	(* Udaljeni rucni ventili; B_x oznake ne odredjuju fizicki identitet. *)
	Act_RV_type : STRUCT (* Udaljeni rucni ventili; B_x fizicki identitet nije potvrdjen. *)
		B_01 : ST_MAN_VALVE; (* Uredjaj/signal oznake B_01. *)
		B_02 : ST_MAN_VALVE; (* Uredjaj/signal oznake B_02. *)
		B_03 : ST_MAN_VALVE; (* Uredjaj/signal oznake B_03. *)
		B_04 : ST_MAN_VALVE; (* Uredjaj/signal oznake B_04. *)
		B_06 : ST_MAN_VALVE; (* Uredjaj/signal oznake B_06. *)
		B_07 : ST_MAN_VALVE; (* Uredjaj/signal oznake B_07. *)
		B_08 : ST_MAN_VALVE; (* Uredjaj/signal oznake B_08. *)
		B_09 : ST_MAN_VALVE; (* Uredjaj/signal oznake B_09. *)
		B_10 : ST_MAN_VALVE; (* Uredjaj/signal oznake B_10. *)
		B_11 : ST_MAN_VALVE; (* Uredjaj/signal oznake B_11. *)
		B_21 : ST_MAN_VALVE; (* Uredjaj/signal oznake B_21. *)
		B_22 : ST_MAN_VALVE; (* Uredjaj/signal oznake B_22. *)
		B_23 : ST_MAN_VALVE; (* Uredjaj/signal oznake B_23. *)
		B_221 : ST_MAN_VALVE; (* Uredjaj/signal oznake B_221. *)
	END_STRUCT;
	(* Udaljeni proporcionalni ventili; B_x oznake ne odredjuju fizicki identitet. *)
	Act_PV_type : STRUCT (* Udaljeni proporcionalni ventili; B_x fizicki identitet nije potvrdjen. *)
		B_01 : ST_VALVE_PV_ACT; (* Uredjaj/signal oznake B_01. *)
		B_201 : ST_VALVE_PV_ACT; (* Uredjaj/signal oznake B_201. *)
	END_STRUCT;
	(* Udaljene pumpe; B_x oznake ne odredjuju fizicki identitet. *)
	Act_Pu_type : STRUCT (* Udaljene pumpe; B_x fizicki identitet nije potvrdjen. *)
		B_101 : ST_PUMP; (* Uredjaj/signal oznake B_101. *)
		B_111 : ST_PUMP; (* Uredjaj/signal oznake B_111. *)
		B_201 : ST_PUMP; (* Uredjaj/signal oznake B_201. *)
		B_211 : ST_PUMP; (* Uredjaj/signal oznake B_211. *)
		B_RB1 : ST_PUMP; (* Uredjaj/signal oznake B_RB1. *)
	END_STRUCT;
	(* Udaljeni automatski ventili; B_x oznake ne odredjuju fizicki identitet. *)
	Act_AV_type : STRUCT (* Udaljeni automatski ventili; B_x fizicki identitet nije potvrdjen. *)
		B_00 : ST_VALVE_ACT_TYPE; (* Uredjaj/signal oznake B_00. *)
		B_02 : ST_VALVE_ACT_TYPE; (* Uredjaj/signal oznake B_02. *)
		B_100 : ST_VALVE_ACT_TYPE; (* Uredjaj/signal oznake B_100. *)
		B_101 : ST_VALVE_ACT_TYPE; (* Uredjaj/signal oznake B_101. *)
		B_102 : ST_VALVE_ACT_TYPE; (* Uredjaj/signal oznake B_102. *)
		B_103 : ST_VALVE_ACT_TYPE; (* Uredjaj/signal oznake B_103. *)
		B_104 : ST_VALVE_ACT_TYPE; (* Uredjaj/signal oznake B_104. *)
		B_105 : ST_VALVE_ACT_TYPE; (* Uredjaj/signal oznake B_105. *)
		B_106 : ST_VALVE_ACT_TYPE; (* Uredjaj/signal oznake B_106. *)
		B_107 : ST_VALVE_ACT_TYPE; (* Uredjaj/signal oznake B_107. *)
		B_108 : ST_VALVE_ACT_TYPE; (* Uredjaj/signal oznake B_108. *)
		B_111 : ST_VALVE_ACT_TYPE; (* Uredjaj/signal oznake B_111. *)
		B_112 : ST_VALVE_ACT_TYPE; (* Uredjaj/signal oznake B_112. *)
		B_113 : ST_VALVE_ACT_TYPE; (* Uredjaj/signal oznake B_113. *)
		B_114 : ST_VALVE_ACT_TYPE; (* Uredjaj/signal oznake B_114. *)
		B_115 : ST_VALVE_ACT_TYPE; (* Uredjaj/signal oznake B_115. *)
		B_116 : ST_VALVE_ACT_TYPE; (* Uredjaj/signal oznake B_116. *)
		B_117 : ST_VALVE_ACT_TYPE; (* Uredjaj/signal oznake B_117. *)
		B_118 : ST_VALVE_ACT_TYPE; (* Uredjaj/signal oznake B_118. *)
		B_200 : ST_VALVE_ACT_TYPE; (* Uredjaj/signal oznake B_200. *)
		B_201 : ST_VALVE_ACT_TYPE; (* Uredjaj/signal oznake B_201. *)
		B_202 : ST_VALVE_ACT_TYPE; (* Uredjaj/signal oznake B_202. *)
		B_203 : ST_VALVE_ACT_TYPE; (* Uredjaj/signal oznake B_203. *)
		B_204 : ST_VALVE_ACT_TYPE; (* Uredjaj/signal oznake B_204. *)
		B_205 : ST_VALVE_ACT_TYPE; (* Uredjaj/signal oznake B_205. *)
		B_211 : ST_VALVE_ACT_TYPE; (* Uredjaj/signal oznake B_211. *)
		B_212 : ST_VALVE_ACT_TYPE; (* Uredjaj/signal oznake B_212. *)
		B_213 : ST_VALVE_ACT_TYPE; (* Uredjaj/signal oznake B_213. *)
		B_214 : ST_VALVE_ACT_TYPE; (* Uredjaj/signal oznake B_214. *)
		B_215 : ST_VALVE_ACT_TYPE; (* Uredjaj/signal oznake B_215. *)
		B_220 : ST_VALVE_ACT_TYPE; (* Uredjaj/signal oznake B_220. *)
		B_301 : ST_VALVE_ACT_TYPE; (* Uredjaj/signal oznake B_301. *)
		B_U22 : ST_VALVE_ACT_TYPE; (* Uredjaj/signal oznake B_U22. *)
		B_U23 : ST_VALVE_ACT_TYPE; (* Uredjaj/signal oznake B_U23. *)
	END_STRUCT;
	(* Zbirna struktura udaljenih IEBKB1 aktuatora. *)
	Act_type : STRUCT (* Zbirna struktura udaljenih IEBKB1 aktuatora. *)
		AV : Act_AV_type; (* Automatski ventili. *)
		RV : Act_RV_type; (* Rucni ventili. *)
		PV : Act_PV_type; (* Proporcionalni ventili. *)
		Pu : Act_Pu_type; (* Pumpe. *)
	END_STRUCT;
	(* Kompletan IEBKB1 komunikacioni snapshot aktuatora, senzora i kontrole. *)
	IEB_KB1_type : STRUCT (* Kompletan IEBKB1 komunikacioni snapshot aktuatora, senzora i kontrole. *)
		Act : Act_type; (* Udaljeni statusi/komande aktuatora. *)
		Sens : Sens_type; (* Senzore i statuse upisuje udaljeni IEBKB1. *)
		Cntrl : Cntrl_type; (* PT/IEBKB1 dvosmerni kontrolni ugovor. *)
	END_STRUCT;
END_TYPE
```

### IEB_KB1_Comm.var - IEBKB1 remote mirror variables
```iecst
VAR
	(* IEBKB1 ogledalo za PT sinoptiku i AsIMA razmenu; ne upravlja lokalnim PT izlazima. *)
	IEB_KB1 : IEB_KB1_type; (* Dvosmerni IEBKB1 snapshot: PT pise zahteve, udaljeni PLC statuse. *)
END_VAR
```

### Package Logical/Libraries - Global libraries

### Library Logical/Libraries/BR_Lib (IEC)
